LIN {X -0.071,Y -362.649,Z 1312.127,A 0.000,B 0.000,C 90.000,E1 238.869} C_DIS
LIN {X -0.108,Y -362.653,Z 1312.127,A 0.000,B 0.000,C 90.000,E1 238.869} C_DIS
LIN {X -0.177,Y -374.472,Z 1312.111,A 0.000,B 0.000,C 90.000,E1 236.087} C_DIS
LIN {X 0.011,Y -387.676,Z 1312.096,A 0.000,B 0.000,C 90.000,E1 233.336} C_DIS
LIN {X 0.004,Y -402.405,Z 1312.082,A 0.000,B 0.000,C 90.000,E1 230.678} C_DIS
LIN {X 0.038,Y -418.775,Z 1312.067,A 0.000,B 0.000,C 90.000,E1 228.081} C_DIS
LIN {X -0.027,Y -436.906,Z 1312.053,A 0.000,B 0.000,C 90.000,E1 225.567} C_DIS
LIN {X -0.154,Y -444.673,Z 1312.048,A 0.000,B 0.000,C 90.000,E1 224.595} C_DIS
LIN {X -0.168,Y -445.603,Z 1312.047,A 0.000,B 0.000,C 90.000,E1 224.433} C_DIS
LIN {X -0.184,Y -446.772,Z 1312.045,A 0.000,B 0.000,C 90.000,E1 224.109} C_DIS
LIN {X -0.199,Y -447.568,Z 1312.043,A 0.000,B 0.000,C 90.000,E1 223.785} C_DIS
LIN {X 0.112,Y -448.651,Z 1312.040,A 0.000,B 0.000,C 90.000,E1 223.095} C_DIS
LIN {X 0.104,Y -449.370,Z 1312.036,A 0.000,B 0.000,C 90.000,E1 222.447} C_DIS
LIN {X -0.202,Y -449.855,Z 1312.032,A 0.000,B 0.000,C 90.000,E1 221.838} C_DIS
LIN {X -0.168,Y -450.246,Z 1312.025,A 0.000,B 0.000,C 90.000,E1 220.539} C_DIS
LIN {X 0.169,Y -452.965,Z 1312.002,A 0.000,B 0.000,C 90.000,E1 216.297} C_DIS
LIN {X -0.050,Y -454.940,Z 1311.989,A 0.000,B 0.000,C 90.000,E1 214.072} C_DIS
LIN {X 0.055,Y -456.951,Z 1311.979,A 0.000,B 0.000,C 90.000,E1 212.133} C_DIS
LIN {X -0.162,Y -460.306,Z 1311.963,A 0.000,B 0.000,C 90.000,E1 209.283} C_DIS
LIN {X 0.239,Y -462.368,Z 1311.954,A 0.000,B 0.000,C 90.000,E1 207.641} C_DIS
LIN {X -0.160,Y -464.683,Z 1311.945,A 0.000,B 0.000,C 90.000,E1 206.104} C_DIS
LIN {X -0.162,Y -467.452,Z 1311.934,A 0.000,B 0.000,C 90.000,E1 204.207} C_DIS
LIN {X -0.141,Y -468.790,Z 1311.929,A 0.000,B 0.000,C 90.000,E1 203.259} C_DIS
LIN {X 0.099,Y -470.556,Z 1311.922,A 0.000,B 0.000,C 90.000,E1 201.972} C_DIS
LIN {X -0.177,Y -473.597,Z 1311.910,A 0.000,B 0.000,C 90.000,E1 199.812} C_DIS
LIN {X 0.200,Y -476.765,Z 1311.898,A 0.000,B 0.000,C 90.000,E1 197.583} C_DIS
LIN {X 0.067,Y -479.940,Z 1311.886,A 0.000,B 0.000,C 90.000,E1 195.426} C_DIS
LIN {X -0.105,Y -482.521,Z 1311.875,A 0.000,B 0.000,C 90.000,E1 193.592} C_DIS
LIN {X 0.143,Y -485.125,Z 1311.865,A 0.000,B 0.000,C 90.000,E1 191.715} C_DIS
LIN {X -0.123,Y -487.671,Z 1311.855,A 0.000,B 0.000,C 90.000,E1 189.905} C_DIS
LIN {X 0.179,Y -489.766,Z 1311.847,A 0.000,B 0.000,C 90.000,E1 188.341} C_DIS
LIN {X 0.034,Y -491.795,Z 1311.838,A 0.000,B 0.000,C 90.000,E1 186.834} C_DIS
LIN {X -0.032,Y -493.392,Z 1311.831,A 0.000,B 0.000,C 90.000,E1 185.625} C_DIS
LIN {X -0.072,Y -494.846,Z 1311.825,A 0.000,B 0.000,C 90.000,E1 184.416} C_DIS
LIN {X -0.240,Y -496.525,Z 1311.816,A 0.000,B 0.000,C 90.000,E1 182.922} C_DIS
LIN {X -0.045,Y -498.194,Z 1311.806,A 0.000,B 0.000,C 90.000,E1 181.088} C_DIS
LIN {X -0.065,Y -499.139,Z 1311.799,A 0.000,B 0.000,C 90.000,E1 179.885} C_DIS
LIN {X -0.197,Y -499.875,Z 1311.791,A 0.000,B 0.000,C 90.000,E1 178.396} C_DIS
LIN {X 0.068,Y -500.147,Z 1311.788,A 0.000,B 0.000,C 90.000,E1 177.764} C_DIS
LIN {X -0.035,Y -500.371,Z 1311.779,A 0.000,B 0.000,C 90.000,E1 176.274} C_DIS
LIN {X 0.114,Y -500.298,Z 1311.774,A 0.000,B 0.000,C 90.000,E1 175.355} C_DIS
LIN {X -0.107,Y -500.165,Z 1311.771,A 0.000,B 0.000,C 90.000,E1 174.780} C_DIS
LIN {X -0.053,Y -499.594,Z 1311.764,A 0.000,B 0.000,C 90.000,E1 173.571} C_DIS
LIN {X 0.133,Y -499.048,Z 1311.759,A 0.000,B 0.000,C 90.000,E1 172.648} C_DIS
LIN {X -0.182,Y -498.189,Z 1311.754,A 0.000,B 0.000,C 90.000,E1 171.781} C_DIS
LIN {X 0.062,Y -496.946,Z 1311.749,A 0.000,B 0.000,C 90.000,E1 170.849} C_DIS
LIN {X 0.211,Y -495.510,Z 1311.744,A 0.000,B 0.000,C 90.000,E1 169.926} C_DIS
LIN {X -0.061,Y -493.810,Z 1311.739,A 0.000,B 0.000,C 90.000,E1 169.050} C_DIS
LIN {X 0.031,Y -490.996,Z 1311.732,A 0.000,B 0.000,C 90.000,E1 167.825} C_DIS
LIN {X -0.073,Y -489.328,Z 1311.729,A 0.000,B 0.000,C 90.000,E1 167.229} C_DIS
LIN {X 0.062,Y -486.673,Z 1311.724,A 0.000,B 0.000,C 90.000,E1 166.297} C_DIS
LIN {X 0.264,Y -482.251,Z 1311.717,A 0.000,B 0.000,C 90.000,E1 165.046} C_DIS
LIN {X 0.175,Y -477.177,Z 1311.711,A 0.000,B 0.000,C 90.000,E1 163.976} C_DIS
LIN {X -0.190,Y -472.157,Z 1311.706,A 0.000,B 0.000,C 90.000,E1 163.087} C_DIS
LIN {X -0.145,Y -463.602,Z 1311.697,A 0.000,B 0.000,C 90.000,E1 161.511} C_DIS
LIN {X -0.178,Y -461.464,Z 1311.695,A 0.000,B 0.000,C 90.000,E1 161.040} C_DIS
LIN {X 0.099,Y -459.056,Z 1311.691,A 0.000,B 0.000,C 90.000,E1 160.369} C_DIS
LIN {X -0.070,Y -457.395,Z 1311.688,A 0.000,B 0.000,C 90.000,E1 159.752} C_DIS
LIN {X -0.080,Y -456.796,Z 1311.683,A 0.000,B 0.000,C 90.000,E1 158.954} C_DIS
LIN {X 0.087,Y -456.802,Z 1311.682,A 0.000,B 0.000,C 90.000,E1 158.773} C_DIS
LIN {X 0.170,Y -457.421,Z 1311.680,A 0.000,B 0.000,C 90.000,E1 158.411} C_DIS
LIN {X 0.130,Y -457.459,Z 1311.680,A 0.000,B 0.000,C 90.000,E1 158.411} C_DIS
LIN {X -0.163,Y -459.940,Z 1311.678,A 0.000,B 0.000,C 90.000,E1 158.103} C_DIS
LIN {X 0.005,Y -463.307,Z 1311.677,A 0.000,B 0.000,C 90.000,E1 157.794} C_DIS
LIN {X -0.102,Y -466.278,Z 1311.675,A 0.000,B 0.000,C 90.000,E1 157.539} C_DIS
LIN {X 0.005,Y -482.916,Z 1311.668,A 0.000,B 0.000,C 90.000,E1 156.177} C_DIS
LIN {X 0.207,Y -490.314,Z 1311.664,A 0.000,B 0.000,C 90.000,E1 155.537} C_DIS
LIN {X 0.022,Y -494.675,Z 1311.662,A 0.000,B 0.000,C 90.000,E1 155.177} C_DIS
LIN {X -0.251,Y -502.876,Z 1311.658,A 0.000,B 0.000,C 90.000,E1 154.409} C_DIS
LIN {X -0.051,Y -506.911,Z 1311.655,A 0.000,B 0.000,C 90.000,E1 153.973} C_DIS
LIN {X 0.132,Y -512.097,Z 1311.652,A 0.000,B 0.000,C 90.000,E1 153.384} C_DIS
LIN {X 0.128,Y -515.865,Z 1311.650,A 0.000,B 0.000,C 90.000,E1 152.948} C_DIS
LIN {X -0.149,Y -519.429,Z 1311.647,A 0.000,B 0.000,C 90.000,E1 152.538} C_DIS
LIN {X -0.104,Y -523.631,Z 1311.644,A 0.000,B 0.000,C 90.000,E1 151.948} C_DIS
LIN {X -0.278,Y -527.388,Z 1311.641,A 0.000,B 0.000,C 90.000,E1 151.385} C_DIS
LIN {X -0.070,Y -531.210,Z 1311.637,A 0.000,B 0.000,C 90.000,E1 150.639} C_DIS
LIN {X -0.201,Y -533.675,Z 1311.634,A 0.000,B 0.000,C 90.000,E1 150.078} C_DIS
LIN {X 0.217,Y -535.635,Z 1311.630,A 0.000,B 0.000,C 90.000,E1 149.459} C_DIS
LIN {X -0.073,Y -536.553,Z 1311.629,A 0.000,B 0.000,C 90.000,E1 149.203} C_DIS
LIN {X 0.093,Y -538.129,Z 1311.626,A 0.000,B 0.000,C 90.000,E1 148.614} C_DIS
LIN {X -0.187,Y -540.015,Z 1311.621,A 0.000,B 0.000,C 90.000,E1 147.788} C_DIS
LIN {X -0.001,Y -541.094,Z 1311.618,A 0.000,B 0.000,C 90.000,E1 147.199} C_DIS
LIN {X 0.052,Y -542.385,Z 1311.613,A 0.000,B 0.000,C 90.000,E1 146.342} C_DIS
LIN {X 0.333,Y -544.220,Z 1311.605,A 0.000,B 0.000,C 90.000,E1 144.895} C_DIS
LIN {X 0.084,Y -544.934,Z 1311.602,A 0.000,B 0.000,C 90.000,E1 144.356} C_DIS
LIN {X -0.181,Y -546.138,Z 1311.599,A 0.000,B 0.000,C 90.000,E1 143.783} C_DIS
LIN {X -0.223,Y -546.147,Z 1311.599,A 0.000,B 0.000,C 90.000,E1 143.783} C_DIS
LIN {X 0.337,Y -546.727,Z 1311.598,A 0.000,B 0.000,C 90.000,E1 143.623} C_DIS
LIN {X 0.195,Y -548.575,Z 1311.597,A 0.000,B 0.000,C 90.000,E1 143.497} C_DIS
LIN {X -0.128,Y -550.841,Z 1311.597,A 0.000,B 0.000,C 90.000,E1 143.417} C_DIS
LIN {X 0.072,Y -560.861,Z 1311.595,A 0.000,B 0.000,C 90.000,E1 143.050} C_DIS
LIN {X 0.300,Y -566.988,Z 1311.593,A 0.000,B 0.000,C 90.000,E1 142.763} C_DIS
LIN {X 0.093,Y -573.111,Z 1311.592,A 0.000,B 0.000,C 90.000,E1 142.477} C_DIS
LIN {X 0.094,Y -580.448,Z 1311.589,A 0.000,B 0.000,C 90.000,E1 142.029} C_DIS
LIN {X 0.232,Y -586.267,Z 1311.587,A 0.000,B 0.000,C 90.000,E1 141.618} C_DIS
LIN {X 0.106,Y -590.462,Z 1311.585,A 0.000,B 0.000,C 90.000,E1 141.295} C_DIS
LIN {X 0.001,Y -594.417,Z 1311.583,A 0.000,B 0.000,C 90.000,E1 140.964} C_DIS
LIN {X -0.084,Y -599.469,Z 1311.580,A 0.000,B 0.000,C 90.000,E1 140.481} C_DIS
LIN {X 0.187,Y -603.081,Z 1311.578,A 0.000,B 0.000,C 90.000,E1 140.070} C_DIS
LIN {X 0.243,Y -607.562,Z 1311.575,A 0.000,B 0.000,C 90.000,E1 139.542} C_DIS
LIN {X -0.207,Y -612.712,Z 1311.572,A 0.000,B 0.000,C 90.000,E1 138.933} C_DIS
LIN {X -0.101,Y -616.473,Z 1311.569,A 0.000,B 0.000,C 90.000,E1 138.405} C_DIS
LIN {X -0.070,Y -620.894,Z 1311.565,A 0.000,B 0.000,C 90.000,E1 137.757} C_DIS
LIN {X 0.083,Y -625.633,Z 1311.561,A 0.000,B 0.000,C 90.000,E1 136.986} C_DIS
LIN {X -0.230,Y -629.505,Z 1311.558,A 0.000,B 0.000,C 90.000,E1 136.377} C_DIS
LIN {X 0.106,Y -636.631,Z 1311.551,A 0.000,B 0.000,C 90.000,E1 135.081} C_DIS
LIN {X -0.085,Y -639.363,Z 1311.548,A 0.000,B 0.000,C 90.000,E1 134.595} C_DIS
LIN {X 0.075,Y -644.084,Z 1311.543,A 0.000,B 0.000,C 90.000,E1 133.704} C_DIS
LIN {X -0.277,Y -651.221,Z 1311.535,A 0.000,B 0.000,C 90.000,E1 132.366} C_DIS
LIN {X 0.029,Y -656.976,Z 1311.529,A 0.000,B 0.000,C 90.000,E1 131.229} C_DIS
LIN {X -0.036,Y -661.842,Z 1311.524,A 0.000,B 0.000,C 90.000,E1 130.253} C_DIS
LIN {X -0.045,Y -666.291,Z 1311.518,A 0.000,B 0.000,C 90.000,E1 129.277} C_DIS
LIN {X -0.004,Y -670.441,Z 1311.513,A 0.000,B 0.000,C 90.000,E1 128.302} C_DIS
LIN {X 0.085,Y -673.306,Z 1311.509,A 0.000,B 0.000,C 90.000,E1 127.569} C_DIS
LIN {X 0.333,Y -676.851,Z 1311.503,A 0.000,B 0.000,C 90.000,E1 126.583} C_DIS
LIN {X 0.083,Y -679.216,Z 1311.499,A 0.000,B 0.000,C 90.000,E1 125.884} C_DIS
LIN {X -0.140,Y -682.074,Z 1311.494,A 0.000,B 0.000,C 90.000,E1 124.945} C_DIS
LIN {X 0.219,Y -684.041,Z 1311.490,A 0.000,B 0.000,C 90.000,E1 124.199} C_DIS
LIN {X -0.341,Y -686.371,Z 1311.485,A 0.000,B 0.000,C 90.000,E1 123.293} C_DIS
LIN {X -0.303,Y -688.375,Z 1311.480,A 0.000,B 0.000,C 90.000,E1 122.339} C_DIS
LIN {X -0.017,Y -690.462,Z 1311.473,A 0.000,B 0.000,C 90.000,E1 121.131} C_DIS
LIN {X -0.283,Y -691.849,Z 1311.468,A 0.000,B 0.000,C 90.000,E1 120.207} C_DIS
LIN {X 0.172,Y -692.835,Z 1311.464,A 0.000,B 0.000,C 90.000,E1 119.461} C_DIS
LIN {X -0.070,Y -693.840,Z 1311.459,A 0.000,B 0.000,C 90.000,E1 118.537} C_DIS
LIN {X -0.016,Y -694.350,Z 1311.453,A 0.000,B 0.000,C 90.000,E1 117.590} C_DIS
LIN {X 0.374,Y -694.631,Z 1311.448,A 0.000,B 0.000,C 90.000,E1 116.616} C_DIS
LIN {X 0.202,Y -694.499,Z 1311.444,A 0.000,B 0.000,C 90.000,E1 115.924} C_DIS
LIN {X 0.079,Y -694.301,Z 1311.442,A 0.000,B 0.000,C 90.000,E1 115.463} C_DIS
LIN {X -0.343,Y -693.843,Z 1311.439,A 0.000,B 0.000,C 90.000,E1 115.027} C_DIS
LIN {X 0.153,Y -693.130,Z 1311.436,A 0.000,B 0.000,C 90.000,E1 114.515} C_DIS
LIN {X 0.113,Y -692.603,Z 1311.435,A 0.000,B 0.000,C 90.000,E1 114.283} C_DIS
LIN {X -0.032,Y -691.135,Z 1311.432,A 0.000,B 0.000,C 90.000,E1 113.823} C_DIS
LIN {X 0.163,Y -688.532,Z 1311.430,A 0.000,B 0.000,C 90.000,E1 113.334} C_DIS
LIN {X 0.277,Y -687.855,Z 1311.429,A 0.000,B 0.000,C 90.000,E1 113.206} C_DIS
LIN {X -0.242,Y -686.910,Z 1311.428,A 0.000,B 0.000,C 90.000,E1 113.131} C_DIS
LIN {X 0.266,Y -681.553,Z 1311.426,A 0.000,B 0.000,C 90.000,E1 112.642} C_DIS
LIN {X -0.175,Y -679.920,Z 1311.425,A 0.000,B 0.000,C 90.000,E1 112.567} C_DIS
LIN {X -0.184,Y -675.396,Z 1311.424,A 0.000,B 0.000,C 90.000,E1 112.386} C_DIS
LIN {X 0.245,Y -673.452,Z 1311.424,A 0.000,B 0.000,C 90.000,E1 112.280} C_DIS
LIN {X -0.220,Y -666.520,Z 1311.423,A 0.000,B 0.000,C 90.000,E1 112.153} C_DIS
LIN {X 0.113,Y -663.945,Z 1311.423,A 0.000,B 0.000,C 90.000,E1 112.078} C_DIS
LIN {X -0.282,Y -655.505,Z 1311.422,A 0.000,B 0.000,C 90.000,E1 112.025} C_DIS
LIN {X 0.065,Y -649.452,Z 1311.422,A 0.000,B 0.000,C 90.000,E1 111.972} C_DIS
LIN {X 0.258,Y -645.085,Z 1311.422,A 0.000,B 0.000,C 90.000,E1 111.897} C_DIS
LIN {X -0.024,Y -643.791,Z 1311.422,A 0.000,B 0.000,C 90.000,E1 111.897} C_DIS
LIN {X -0.078,Y -642.090,Z 1311.421,A 0.000,B 0.000,C 90.000,E1 111.844} C_DIS
LIN {X -0.119,Y -642.053,Z 1311.421,A 0.000,B 0.000,C 90.000,E1 111.844} C_DIS
LIN {X -0.156,Y -643.053,Z 1311.420,A 0.000,B 0.000,C 90.000,E1 111.642} C_DIS
LIN {X 0.244,Y -645.869,Z 1311.418,A 0.000,B 0.000,C 90.000,E1 111.227} C_DIS
LIN {X 0.229,Y -651.693,Z 1311.414,A 0.000,B 0.000,C 90.000,E1 110.482} C_DIS
LIN {X -0.008,Y -655.900,Z 1311.411,A 0.000,B 0.000,C 90.000,E1 109.885} C_DIS
LIN {X 0.015,Y -659.535,Z 1311.407,A 0.000,B 0.000,C 90.000,E1 109.268} C_DIS
LIN {X -0.153,Y -662.652,Z 1311.404,A 0.000,B 0.000,C 90.000,E1 108.671} C_DIS
LIN {X -0.237,Y -665.922,Z 1311.400,A 0.000,B 0.000,C 90.000,E1 107.946} C_DIS
LIN {X -0.294,Y -668.770,Z 1311.396,A 0.000,B 0.000,C 90.000,E1 107.221} C_DIS
LIN {X -0.254,Y -670.453,Z 1311.393,A 0.000,B 0.000,C 90.000,E1 106.732} C_DIS
LIN {X 0.183,Y -672.621,Z 1311.389,A 0.000,B 0.000,C 90.000,E1 105.969} C_DIS
LIN {X 0.183,Y -674.414,Z 1311.385,A 0.000,B 0.000,C 90.000,E1 105.245} C_DIS
LIN {X 0.018,Y -675.919,Z 1311.381,A 0.000,B 0.000,C 90.000,E1 104.537} C_DIS
LIN {X -0.131,Y -677.197,Z 1311.377,A 0.000,B 0.000,C 90.000,E1 103.828} C_DIS
LIN {X -0.269,Y -677.981,Z 1311.373,A 0.000,B 0.000,C 90.000,E1 103.119} C_DIS
LIN {X 0.260,Y -678.463,Z 1311.369,A 0.000,B 0.000,C 90.000,E1 102.355} C_DIS
LIN {X 0.171,Y -678.639,Z 1311.366,A 0.000,B 0.000,C 90.000,E1 101.883} C_DIS
LIN {X -0.053,Y -678.589,Z 1311.364,A 0.000,B 0.000,C 90.000,E1 101.422} C_DIS
LIN {X -0.188,Y -678.054,Z 1311.359,A 0.000,B 0.000,C 90.000,E1 100.715} C_DIS
LIN {X 0.259,Y -677.529,Z 1311.357,A 0.000,B 0.000,C 90.000,E1 100.197} C_DIS
LIN {X 0.156,Y -676.732,Z 1311.354,A 0.000,B 0.000,C 90.000,E1 99.726} C_DIS
LIN {X -0.068,Y -675.668,Z 1311.351,A 0.000,B 0.000,C 90.000,E1 99.265} C_DIS
LIN {X -0.292,Y -674.222,Z 1311.349,A 0.000,B 0.000,C 90.000,E1 98.803} C_DIS
LIN {X 0.072,Y -671.486,Z 1311.345,A 0.000,B 0.000,C 90.000,E1 98.049} C_DIS
LIN {X -0.258,Y -668.089,Z 1311.341,A 0.000,B 0.000,C 90.000,E1 97.352} C_DIS
LIN {X 0.135,Y -665.537,Z 1311.338,A 0.000,B 0.000,C 90.000,E1 96.834} C_DIS
LIN {X -0.336,Y -661.432,Z 1311.334,A 0.000,B 0.000,C 90.000,E1 96.144} C_DIS
LIN {X -0.087,Y -657.553,Z 1311.331,A 0.000,B 0.000,C 90.000,E1 95.511} C_DIS
LIN {X 0.128,Y -653.294,Z 1311.327,A 0.000,B 0.000,C 90.000,E1 94.878} C_DIS
LIN {X -0.235,Y -649.570,Z 1311.324,A 0.000,B 0.000,C 90.000,E1 94.416} C_DIS
LIN {X -0.091,Y -644.408,Z 1311.321,A 0.000,B 0.000,C 90.000,E1 93.784} C_DIS
LIN {X -0.030,Y -638.855,Z 1311.318,A 0.000,B 0.000,C 90.000,E1 93.154} C_DIS
LIN {X -0.094,Y -631.872,Z 1311.313,A 0.000,B 0.000,C 90.000,E1 92.407} C_DIS
LIN {X 0.015,Y -625.689,Z 1311.310,A 0.000,B 0.000,C 90.000,E1 91.776} C_DIS
LIN {X -0.275,Y -620.348,Z 1311.307,A 0.000,B 0.000,C 90.000,E1 91.318} C_DIS
LIN {X 0.254,Y -616.296,Z 1311.305,A 0.000,B 0.000,C 90.000,E1 90.917} C_DIS
LIN {X 0.010,Y -608.830,Z 1311.302,A 0.000,B 0.000,C 90.000,E1 90.401} C_DIS
LIN {X 0.226,Y -602.513,Z 1311.300,A 0.000,B 0.000,C 90.000,E1 90.000} C_DIS
LIN {X 0.163,Y -595.886,Z 1311.298,A 0.000,B 0.000,C 90.000,E1 89.656} C_DIS
LIN {X -0.081,Y -588.867,Z 1311.297,A 0.000,B 0.000,C 90.000,E1 89.370} C_DIS
LIN {X -0.101,Y -576.659,Z 1311.294,A 0.000,B 0.000,C 90.000,E1 88.912} C_DIS
LIN {X -0.178,Y -572.876,Z 1311.293,A 0.000,B 0.000,C 90.000,E1 88.740} C_DIS
LIN {X -0.217,Y -572.799,Z 1311.293,A 0.000,B 0.000,C 90.000,E1 88.740} C_DIS
LIN {X 0.199,Y -570.811,Z 1311.292,A 0.000,B 0.000,C 90.000,E1 88.453} C_DIS
LIN {X 0.156,Y -570.803,Z 1311.292,A 0.000,B 0.000,C 90.000,E1 88.453} C_DIS
LIN {X 0.144,Y -570.501,Z 1311.290,A 0.000,B 0.000,C 90.000,E1 88.224} C_DIS
LIN {X 0.053,Y -570.697,Z 1311.287,A 0.000,B 0.000,C 90.000,E1 87.650} C_DIS
LIN {X 0.035,Y -571.783,Z 1311.281,A 0.000,B 0.000,C 90.000,E1 86.560} C_DIS
LIN {X -0.173,Y -574.648,Z 1311.266,A 0.000,B 0.000,C 90.000,E1 83.856} C_DIS
LIN {X 0.204,Y -577.511,Z 1311.252,A 0.000,B 0.000,C 90.000,E1 81.376} C_DIS
LIN {X 0.264,Y -579.450,Z 1311.243,A 0.000,B 0.000,C 90.000,E1 79.746} C_DIS
LIN {X 0.136,Y -580.891,Z 1311.236,A 0.000,B 0.000,C 90.000,E1 78.409} C_DIS
LIN {X -0.194,Y -582.408,Z 1311.227,A 0.000,B 0.000,C 90.000,E1 76.825} C_DIS
LIN {X -0.025,Y -583.440,Z 1311.219,A 0.000,B 0.000,C 90.000,E1 75.463} C_DIS
LIN {X -0.068,Y -584.221,Z 1311.213,A 0.000,B 0.000,C 90.000,E1 74.393} C_DIS
LIN {X 0.127,Y -585.071,Z 1311.206,A 0.000,B 0.000,C 90.000,E1 73.032} C_DIS
LIN {X -0.207,Y -586.113,Z 1311.197,A 0.000,B 0.000,C 90.000,E1 71.456} C_DIS
LIN {X 0.040,Y -587.148,Z 1311.188,A 0.000,B 0.000,C 90.000,E1 69.826} C_DIS
LIN {X -0.048,Y -588.218,Z 1311.179,A 0.000,B 0.000,C 90.000,E1 68.230} C_DIS
LIN {X -0.319,Y -589.132,Z 1311.172,A 0.000,B 0.000,C 90.000,E1 66.922} C_DIS
LIN {X -0.006,Y -590.407,Z 1311.161,A 0.000,B 0.000,C 90.000,E1 65.025} C_DIS
LIN {X -0.187,Y -591.697,Z 1311.151,A 0.000,B 0.000,C 90.000,E1 63.179} C_DIS
LIN {X -0.172,Y -593.530,Z 1311.139,A 0.000,B 0.000,C 90.000,E1 61.051} C_DIS
LIN {X -0.046,Y -595.600,Z 1311.127,A 0.000,B 0.000,C 90.000,E1 58.918} C_DIS
LIN {X 0.227,Y -597.569,Z 1311.117,A 0.000,B 0.000,C 90.000,E1 57.041} C_DIS
LIN {X -0.110,Y -598.989,Z 1311.110,A 0.000,B 0.000,C 90.000,E1 55.754} C_DIS
LIN {X 0.009,Y -600.062,Z 1311.104,A 0.000,B 0.000,C 90.000,E1 54.689} C_DIS
LIN {X -0.195,Y -601.500,Z 1311.095,A 0.000,B 0.000,C 90.000,E1 53.130} C_DIS
LIN {X -0.009,Y -602.810,Z 1311.086,A 0.000,B 0.000,C 90.000,E1 51.537} C_DIS
LIN {X -0.019,Y -604.099,Z 1311.076,A 0.000,B 0.000,C 90.000,E1 49.703} C_DIS
LIN {X -0.178,Y -604.564,Z 1311.072,A 0.000,B 0.000,C 90.000,E1 48.933} C_DIS
LIN {X -0.079,Y -604.890,Z 1311.066,A 0.000,B 0.000,C 90.000,E1 47.877} C_DIS
LIN {X -0.160,Y -605.118,Z 1311.056,A 0.000,B 0.000,C 90.000,E1 46.053} C_DIS
LIN {X -0.082,Y -605.165,Z 1311.050,A 0.000,B 0.000,C 90.000,E1 45.000} C_DIS
LIN {X -0.003,Y -605.019,Z 1311.044,A 0.000,B 0.000,C 90.000,E1 43.947} C_DIS
LIN {X 0.113,Y -604.567,Z 1311.036,A 0.000,B 0.000,C 90.000,E1 42.366} C_DIS
LIN {X 0.011,Y -604.123,Z 1311.028,A 0.000,B 0.000,C 90.000,E1 41.067} C_DIS
LIN {X 0.107,Y -603.633,Z 1311.022,A 0.000,B 0.000,C 90.000,E1 40.011} C_DIS
LIN {X -0.188,Y -603.162,Z 1311.017,A 0.000,B 0.000,C 90.000,E1 38.991} C_DIS
LIN {X 0.107,Y -602.673,Z 1311.012,A 0.000,B 0.000,C 90.000,E1 38.177} C_DIS
LIN {X 0.026,Y -602.049,Z 1311.008,A 0.000,B 0.000,C 90.000,E1 37.397} C_DIS
LIN {X -0.288,Y -600.957,Z 1311.002,A 0.000,B 0.000,C 90.000,E1 36.377} C_DIS
LIN {X 0.104,Y -599.106,Z 1310.995,A 0.000,B 0.000,C 90.000,E1 35.025} C_DIS
LIN {X -0.119,Y -597.290,Z 1310.989,A 0.000,B 0.000,C 90.000,E1 33.992} C_DIS
LIN {X 0.238,Y -595.709,Z 1310.984,A 0.000,B 0.000,C 90.000,E1 33.166} C_DIS
LIN {X -0.246,Y -593.925,Z 1310.980,A 0.000,B 0.000,C 90.000,E1 32.418} C_DIS
LIN {X 0.070,Y -591.876,Z 1310.976,A 0.000,B 0.000,C 90.000,E1 31.592} C_DIS
LIN {X 0.051,Y -589.439,Z 1310.971,A 0.000,B 0.000,C 90.000,E1 30.797} C_DIS
LIN {X 0.125,Y -587.679,Z 1310.968,A 0.000,B 0.000,C 90.000,E1 30.256} C_DIS
LIN {X 0.062,Y -584.645,Z 1310.964,A 0.000,B 0.000,C 90.000,E1 29.461} C_DIS
LIN {X -0.186,Y -582.373,Z 1310.961,A 0.000,B 0.000,C 90.000,E1 28.949} C_DIS
LIN {X 0.205,Y -578.708,Z 1310.956,A 0.000,B 0.000,C 90.000,E1 28.103} C_DIS
LIN {X 0.038,Y -574.503,Z 1310.952,A 0.000,B 0.000,C 90.000,E1 27.308} C_DIS
LIN {X 0.153,Y -570.702,Z 1310.948,A 0.000,B 0.000,C 90.000,E1 26.616} C_DIS
LIN {X 0.153,Y -565.727,Z 1310.943,A 0.000,B 0.000,C 90.000,E1 25.796} C_DIS
LIN {X -0.308,Y -561.156,Z 1310.940,A 0.000,B 0.000,C 90.000,E1 25.155} C_DIS
LIN {X -0.096,Y -558.238,Z 1310.937,A 0.000,B 0.000,C 90.000,E1 24.719} C_DIS
LIN {X -0.112,Y -552.956,Z 1310.933,A 0.000,B 0.000,C 90.000,E1 24.027} C_DIS
LIN {X -0.166,Y -547.401,Z 1310.930,A 0.000,B 0.000,C 90.000,E1 23.334} C_DIS
LIN {X 0.098,Y -540.177,Z 1310.925,A 0.000,B 0.000,C 90.000,E1 22.461} C_DIS
LIN {X -0.085,Y -533.890,Z 1310.921,A 0.000,B 0.000,C 90.000,E1 21.770} C_DIS
LIN {X 0.239,Y -522.221,Z 1310.914,A 0.000,B 0.000,C 90.000,E1 20.482} C_DIS
LIN {X 0.115,Y -512.971,Z 1310.909,A 0.000,B 0.000,C 90.000,E1 19.523} C_DIS
LIN {X 0.023,Y -501.882,Z 1310.902,A 0.000,B 0.000,C 90.000,E1 18.417} C_DIS
LIN {X 0.151,Y -490.858,Z 1310.896,A 0.000,B 0.000,C 90.000,E1 17.330} C_DIS
LIN {X -0.160,Y -483.700,Z 1310.893,A 0.000,B 0.000,C 90.000,E1 16.677} C_DIS
LIN {X 0.078,Y -476.334,Z 1310.889,A 0.000,B 0.000,C 90.000,E1 15.969} C_DIS
LIN {X 0.109,Y -464.557,Z 1310.883,A 0.000,B 0.000,C 90.000,E1 14.898} C_DIS
LIN {X -0.185,Y -442.753,Z 1310.871,A 0.000,B 0.000,C 90.000,E1 12.883} C_DIS
LIN {X -0.129,Y -424.029,Z 1310.861,A 0.000,B 0.000,C 90.000,E1 10.950} C_DIS
LIN {X 0.003,Y -409.779,Z 1310.852,A 0.000,B 0.000,C 90.000,E1 9.378} C_DIS
LIN {X 0.171,Y -401.165,Z 1310.847,A 0.000,B 0.000,C 90.000,E1 8.398} C_DIS
LIN {X -0.089,Y -398.370,Z 1310.845,A 0.000,B 0.000,C 90.000,E1 8.106} C_DIS
LIN {X -0.074,Y -395.420,Z 1310.842,A 0.000,B 0.000,C 90.000,E1 7.644} C_DIS
LIN {X -0.112,Y -395.442,Z 1310.842,A 0.000,B 0.000,C 90.000,E1 7.644} C_DIS
LIN {X 0.154,Y -396.271,Z 1310.842,A 0.000,B 0.000,C 90.000,E1 7.473} C_DIS
LIN {X 0.018,Y -400.435,Z 1310.840,A 0.000,B 0.000,C 90.000,E1 7.125} C_DIS
LIN {X 0.136,Y -408.992,Z 1310.837,A 0.000,B 0.000,C 90.000,E1 6.549} C_DIS
LIN {X 0.088,Y -417.236,Z 1310.834,A 0.000,B 0.000,C 90.000,E1 6.030} C_DIS
LIN {X 0.145,Y -423.721,Z 1310.831,A 0.000,B 0.000,C 90.000,E1 5.568} C_DIS
LIN {X -0.158,Y -433.047,Z 1310.827,A 0.000,B 0.000,C 90.000,E1 4.878} C_DIS
LIN {X 0.123,Y -442.041,Z 1310.823,A 0.000,B 0.000,C 90.000,E1 4.073} C_DIS
LIN {X -0.030,Y -450.911,Z 1310.818,A 0.000,B 0.000,C 90.000,E1 3.269} C_DIS
LIN {X 0.227,Y -458.153,Z 1310.814,A 0.000,B 0.000,C 90.000,E1 2.522} C_DIS
LIN {X -0.029,Y -462.248,Z 1310.812,A 0.000,B 0.000,C 90.000,E1 2.121} C_DIS
LIN {X 0.088,Y -466.383,Z 1310.809,A 0.000,B 0.000,C 90.000,E1 1.661} C_DIS
LIN {X 0.194,Y -472.544,Z 1310.805,A 0.000,B 0.000,C 90.000,E1 0.917} C_DIS
LIN {X -0.084,Y -478.505,Z 1310.801,A 0.000,B 0.000,C 90.000,E1 0.172} C_DIS
LIN {X 0.138,Y -484.372,Z 1310.796,A 0.000,B 0.000,C 90.000,E1 359.312} C_DIS
LIN {X -0.062,Y -489.328,Z 1310.792,A 0.000,B 0.000,C 90.000,E1 358.568} C_DIS
LIN {X -0.202,Y -493.919,Z 1310.788,A 0.000,B 0.000,C 90.000,E1 357.822} C_DIS
LIN {X -0.001,Y -497.459,Z 1310.784,A 0.000,B 0.000,C 90.000,E1 357.192} C_DIS
LIN {X 0.124,Y -502.221,Z 1310.779,A 0.000,B 0.000,C 90.000,E1 356.274} C_DIS
LIN {X 0.109,Y -505.946,Z 1310.775,A 0.000,B 0.000,C 90.000,E1 355.527} C_DIS
LIN {X 0.130,Y -509.406,Z 1310.771,A 0.000,B 0.000,C 90.000,E1 354.780} C_DIS
LIN {X 0.139,Y -513.978,Z 1310.765,A 0.000,B 0.000,C 90.000,E1 353.742} C_DIS
LIN {X 0.013,Y -516.372,Z 1310.762,A 0.000,B 0.000,C 90.000,E1 353.166} C_DIS
LIN {X -0.115,Y -519.623,Z 1310.757,A 0.000,B 0.000,C 90.000,E1 352.299} C_DIS
LIN {X -0.210,Y -522.596,Z 1310.752,A 0.000,B 0.000,C 90.000,E1 351.432} C_DIS
LIN {X -0.202,Y -524.397,Z 1310.749,A 0.000,B 0.000,C 90.000,E1 350.849} C_DIS
LIN {X -0.228,Y -527.751,Z 1310.743,A 0.000,B 0.000,C 90.000,E1 349.690} C_DIS
LIN {X -0.148,Y -530.014,Z 1310.738,A 0.000,B 0.000,C 90.000,E1 348.814} C_DIS
LIN {X -0.079,Y -531.373,Z 1310.735,A 0.000,B 0.000,C 90.000,E1 348.229} C_DIS
LIN {X 0.086,Y -533.805,Z 1310.728,A 0.000,B 0.000,C 90.000,E1 347.061} C_DIS
LIN {X -0.168,Y -535.311,Z 1310.723,A 0.000,B 0.000,C 90.000,E1 346.228} C_DIS
LIN {X 0.178,Y -537.055,Z 1310.717,A 0.000,B 0.000,C 90.000,E1 345.046} C_DIS
LIN {X -0.231,Y -537.771,Z 1310.714,A 0.000,B 0.000,C 90.000,E1 344.519} C_DIS
LIN {X -0.229,Y -538.712,Z 1310.708,A 0.000,B 0.000,C 90.000,E1 343.378} C_DIS
LIN {X 0.092,Y -539.315,Z 1310.703,A 0.000,B 0.000,C 90.000,E1 342.489} C_DIS
LIN {X 0.066,Y -539.488,Z 1310.698,A 0.000,B 0.000,C 90.000,E1 341.638} C_DIS
LIN {X -0.196,Y -539.132,Z 1310.690,A 0.000,B 0.000,C 90.000,E1 340.242} C_DIS
LIN {X 0.065,Y -538.772,Z 1310.687,A 0.000,B 0.000,C 90.000,E1 339.645} C_DIS
LIN {X 0.225,Y -537.970,Z 1310.682,A 0.000,B 0.000,C 90.000,E1 338.773} C_DIS
LIN {X 0.183,Y -536.943,Z 1310.677,A 0.000,B 0.000,C 90.000,E1 337.922} C_DIS
LIN {X 0.117,Y -536.085,Z 1310.674,A 0.000,B 0.000,C 90.000,E1 337.358} C_DIS
LIN {X 0.047,Y -534.907,Z 1310.671,A 0.000,B 0.000,C 90.000,E1 336.794} C_DIS
LIN {X -0.168,Y -534.482,Z 1310.670,A 0.000,B 0.000,C 90.000,E1 336.538} C_DIS
LIN {X -0.045,Y -532.331,Z 1310.665,A 0.000,B 0.000,C 90.000,E1 335.665} C_DIS
LIN {X 0.049,Y -529.897,Z 1310.660,A 0.000,B 0.000,C 90.000,E1 334.793} C_DIS
LIN {X -0.105,Y -524.390,Z 1310.650,A 0.000,B 0.000,C 90.000,E1 333.076} C_DIS
LIN {X 0.044,Y -520.538,Z 1310.644,A 0.000,B 0.000,C 90.000,E1 331.897} C_DIS
LIN {X -0.229,Y -517.521,Z 1310.639,A 0.000,B 0.000,C 90.000,E1 331.051} C_DIS
LIN {X 0.169,Y -514.299,Z 1310.634,A 0.000,B 0.000,C 90.000,E1 330.127} C_DIS
LIN {X 0.002,Y -511.402,Z 1310.630,A 0.000,B 0.000,C 90.000,E1 329.410} C_DIS
LIN {X 0.104,Y -505.146,Z 1310.622,A 0.000,B 0.000,C 90.000,E1 327.916} C_DIS
LIN {X 0.017,Y -499.499,Z 1310.614,A 0.000,B 0.000,C 90.000,E1 326.580} C_DIS
LIN {X -0.235,Y -497.281,Z 1310.611,A 0.000,B 0.000,C 90.000,E1 326.008} C_DIS
LIN {X -0.090,Y -495.617,Z 1310.608,A 0.000,B 0.000,C 90.000,E1 325.388} C_DIS
LIN {X -0.102,Y -493.843,Z 1310.603,A 0.000,B 0.000,C 90.000,E1 324.482} C_DIS
LIN {X 0.010,Y -492.369,Z 1310.596,A 0.000,B 0.000,C 90.000,E1 323.256} C_DIS
LIN {X 0.103,Y -491.341,Z 1310.589,A 0.000,B 0.000,C 90.000,E1 322.029} C_DIS
LIN {X 0.025,Y -490.436,Z 1310.584,A 0.000,B 0.000,C 90.000,E1 321.126} C_DIS
LIN {X 0.018,Y -489.633,Z 1310.581,A 0.000,B 0.000,C 90.000,E1 320.517} C_DIS
LIN {X 0.169,Y -489.102,Z 1310.579,A 0.000,B 0.000,C 90.000,E1 320.194} C_DIS
LIN {X 0.007,Y -488.432,Z 1310.577,A 0.000,B 0.000,C 90.000,E1 319.908} C_DIS
LIN {X -0.158,Y -487.555,Z 1310.576,A 0.000,B 0.000,C 90.000,E1 319.622} C_DIS
LIN {X -0.083,Y -486.987,Z 1310.575,A 0.000,B 0.000,C 90.000,E1 319.461} C_DIS
LIN {X -0.009,Y -486.260,Z 1310.574,A 0.000,B 0.000,C 90.000,E1 319.299} C_DIS
LIN {X 0.064,Y -485.175,Z 1310.573,A 0.000,B 0.000,C 90.000,E1 319.138} C_DIS
LIN {X 0.171,Y -463.298,Z 1310.560,A 0.000,B 0.000,C 90.000,E1 316.782} C_DIS
LIN {X -0.012,Y -443.766,Z 1310.547,A 0.000,B 0.000,C 90.000,E1 314.433} C_DIS
LIN {X -0.052,Y -425.796,Z 1310.533,A 0.000,B 0.000,C 90.000,E1 311.962} C_DIS
LIN {X 0.054,Y -409.544,Z 1310.519,A 0.000,B 0.000,C 90.000,E1 309.402} C_DIS
LIN {X 0.064,Y -394.887,Z 1310.505,A 0.000,B 0.000,C 90.000,E1 306.790} C_DIS
LIN {X -0.154,Y -389.671,Z 1310.499,A 0.000,B 0.000,C 90.000,E1 305.804} C_DIS
LIN {X -0.191,Y -389.672,Z 1310.499,A 0.000,B 0.000,C 90.000,E1 305.804} C_DIS
LIN {X 0.037,Y -391.347,Z 1310.492,A 0.000,B 0.000,C 90.000,E1 304.485} C_DIS
LIN {X -0.140,Y -397.058,Z 1310.458,A 0.000,B 0.000,C 90.000,E1 298.487} C_DIS
LIN {X 0.165,Y -401.450,Z 1310.427,A 0.000,B 0.000,C 90.000,E1 292.823} C_DIS
LIN {X -0.125,Y -401.677,Z 1310.425,A 0.000,B 0.000,C 90.000,E1 292.514} C_DIS
LIN {X -0.095,Y -404.537,Z 1310.396,A 0.000,B 0.000,C 90.000,E1 287.275} C_DIS
LIN {X 0.005,Y -404.763,Z 1310.394,A 0.000,B 0.000,C 90.000,E1 286.913} C_DIS
LIN {X -0.088,Y -406.150,Z 1310.363,A 0.000,B 0.000,C 90.000,E1 281.366} C_DIS
LIN {X 0.017,Y -405.648,Z 1310.334,A 0.000,B 0.000,C 90.000,E1 276.144} C_DIS
LIN {X 0.021,Y -405.625,Z 1310.332,A 0.000,B 0.000,C 90.000,E1 275.796} C_DIS
LIN {X 0.094,Y -403.554,Z 1310.305,A 0.000,B 0.000,C 90.000,E1 270.917} C_DIS
LIN {X 0.029,Y -403.075,Z 1310.301,A 0.000,B 0.000,C 90.000,E1 270.229} C_DIS
LIN {X -0.144,Y -399.024,Z 1310.272,A 0.000,B 0.000,C 90.000,E1 265.008} C_DIS
LIN {X 0.169,Y -398.149,Z 1310.268,A 0.000,B 0.000,C 90.000,E1 264.261} C_DIS
LIN {X 0.027,Y -392.946,Z 1310.241,A 0.000,B 0.000,C 90.000,E1 259.342} C_DIS
LIN {X -0.015,Y -392.509,Z 1310.239,A 0.000,B 0.000,C 90.000,E1 258.993} C_DIS
LIN {X 0.132,Y -386.143,Z 1310.213,A 0.000,B 0.000,C 90.000,E1 254.338} C_DIS
LIN {X 0.093,Y -385.021,Z 1310.207,A 0.000,B 0.000,C 90.000,E1 253.268} C_DIS
LIN {X -0.034,Y -378.157,Z 1310.183,A 0.000,B 0.000,C 90.000,E1 248.954} C_DIS
LIN {X 0.179,Y -375.917,Z 1310.173,A 0.000,B 0.000,C 90.000,E1 247.102} C_DIS
LIN {X -0.201,Y -369.131,Z 1310.151,A 0.000,B 0.000,C 90.000,E1 243.127} C_DIS
LIN {X 0.028,Y -366.281,Z 1310.138,A 0.000,B 0.000,C 90.000,E1 240.873} C_DIS
LIN {X -0.002,Y -365.045,Z 1310.135,A 0.000,B 0.000,C 90.000,E1 240.205} C_DIS
LIN {X -0.040,Y -365.050,Z 1310.135,A 0.000,B 0.000,C 90.000,E1 240.205} C_DIS
LIN {X -0.054,Y -376.507,Z 1310.119,A 0.000,B 0.000,C 90.000,E1 237.375} C_DIS
LIN {X 0.074,Y -389.097,Z 1310.104,A 0.000,B 0.000,C 90.000,E1 234.642} C_DIS
LIN {X 0.104,Y -403.152,Z 1310.089,A 0.000,B 0.000,C 90.000,E1 231.984} C_DIS
LIN {X 0.206,Y -418.776,Z 1310.075,A 0.000,B 0.000,C 90.000,E1 229.380} C_DIS
LIN {X -0.155,Y -436.080,Z 1310.061,A 0.000,B 0.000,C 90.000,E1 226.905} C_DIS
LIN {X 0.010,Y -444.768,Z 1310.054,A 0.000,B 0.000,C 90.000,E1 225.729} C_DIS
LIN {X -0.001,Y -445.877,Z 1310.053,A 0.000,B 0.000,C 90.000,E1 225.567} C_DIS
LIN {X -0.011,Y -446.609,Z 1310.052,A 0.000,B 0.000,C 90.000,E1 225.405} C_DIS
LIN {X -0.023,Y -447.612,Z 1310.051,A 0.000,B 0.000,C 90.000,E1 225.081} C_DIS
LIN {X -0.032,Y -448.325,Z 1310.049,A 0.000,B 0.000,C 90.000,E1 224.757} C_DIS
LIN {X -0.040,Y -449.296,Z 1310.045,A 0.000,B 0.000,C 90.000,E1 224.109} C_DIS
LIN {X -0.040,Y -449.902,Z 1310.042,A 0.000,B 0.000,C 90.000,E1 223.461} C_DIS
LIN {X -0.010,Y -450.429,Z 1310.036,A 0.000,B 0.000,C 90.000,E1 222.486} C_DIS
LIN {X -0.001,Y -450.643,Z 1310.031,A 0.000,B 0.000,C 90.000,E1 221.515} C_DIS
LIN {X -0.078,Y -452.229,Z 1310.011,A 0.000,B 0.000,C 90.000,E1 217.971} C_DIS
LIN {X -0.224,Y -453.515,Z 1310.002,A 0.000,B 0.000,C 90.000,E1 216.377} C_DIS
LIN {X 0.108,Y -455.190,Z 1309.991,A 0.000,B 0.000,C 90.000,E1 214.405} C_DIS
LIN {X 0.082,Y -457.472,Z 1309.979,A 0.000,B 0.000,C 90.000,E1 212.163} C_DIS
LIN {X -0.150,Y -461.246,Z 1309.961,A 0.000,B 0.000,C 90.000,E1 208.999} C_DIS
LIN {X 0.021,Y -464.762,Z 1309.947,A 0.000,B 0.000,C 90.000,E1 206.437} C_DIS
LIN {X 0.110,Y -468.457,Z 1309.933,A 0.000,B 0.000,C 90.000,E1 203.898} C_DIS
LIN {X -0.036,Y -471.478,Z 1309.921,A 0.000,B 0.000,C 90.000,E1 201.716} C_DIS
LIN {X 0.183,Y -474.148,Z 1309.910,A 0.000,B 0.000,C 90.000,E1 199.812} C_DIS
LIN {X 0.122,Y -477.362,Z 1309.898,A 0.000,B 0.000,C 90.000,E1 197.638} C_DIS
LIN {X -0.152,Y -481.027,Z 1309.884,A 0.000,B 0.000,C 90.000,E1 195.190} C_DIS
LIN {X 0.173,Y -483.658,Z 1309.874,A 0.000,B 0.000,C 90.000,E1 193.300} C_DIS
LIN {X -0.027,Y -486.304,Z 1309.864,A 0.000,B 0.000,C 90.000,E1 191.478} C_DIS
LIN {X 0.211,Y -488.873,Z 1309.854,A 0.000,B 0.000,C 90.000,E1 189.613} C_DIS
LIN {X -0.063,Y -491.421,Z 1309.843,A 0.000,B 0.000,C 90.000,E1 187.814} C_DIS
LIN {X 0.244,Y -493.496,Z 1309.835,A 0.000,B 0.000,C 90.000,E1 186.258} C_DIS
LIN {X 0.097,Y -495.452,Z 1309.827,A 0.000,B 0.000,C 90.000,E1 184.759} C_DIS
LIN {X 0.046,Y -496.864,Z 1309.820,A 0.000,B 0.000,C 90.000,E1 183.555} C_DIS
LIN {X 0.157,Y -497.858,Z 1309.815,A 0.000,B 0.000,C 90.000,E1 182.636} C_DIS
LIN {X 0.015,Y -499.295,Z 1309.806,A 0.000,B 0.000,C 90.000,E1 181.146} C_DIS
LIN {X 0.012,Y -500.298,Z 1309.800,A 0.000,B 0.000,C 90.000,E1 179.943} C_DIS
LIN {X -0.098,Y -501.194,Z 1309.791,A 0.000,B 0.000,C 90.000,E1 178.453} C_DIS
LIN {X 0.058,Y -501.611,Z 1309.786,A 0.000,B 0.000,C 90.000,E1 177.535} C_DIS
LIN {X -0.021,Y -501.901,Z 1309.778,A 0.000,B 0.000,C 90.000,E1 176.045} C_DIS
LIN {X 0.185,Y -501.869,Z 1309.773,A 0.000,B 0.000,C 90.000,E1 175.122} C_DIS
LIN {X -0.149,Y -501.633,Z 1309.768,A 0.000,B 0.000,C 90.000,E1 174.261} C_DIS
LIN {X -0.150,Y -500.963,Z 1309.760,A 0.000,B 0.000,C 90.000,E1 172.761} C_DIS
LIN {X -0.023,Y -499.917,Z 1309.753,A 0.000,B 0.000,C 90.000,E1 171.546} C_DIS
LIN {X 0.163,Y -498.797,Z 1309.748,A 0.000,B 0.000,C 90.000,E1 170.622} C_DIS
LIN {X -0.073,Y -497.349,Z 1309.743,A 0.000,B 0.000,C 90.000,E1 169.746} C_DIS
LIN {X 0.164,Y -495.722,Z 1309.738,A 0.000,B 0.000,C 90.000,E1 168.814} C_DIS
LIN {X 0.187,Y -492.224,Z 1309.730,A 0.000,B 0.000,C 90.000,E1 167.297} C_DIS
LIN {X -0.011,Y -489.652,Z 1309.724,A 0.000,B 0.000,C 90.000,E1 166.408} C_DIS
LIN {X -0.115,Y -487.898,Z 1309.721,A 0.000,B 0.000,C 90.000,E1 165.811} C_DIS
LIN {X -0.009,Y -483.612,Z 1309.714,A 0.000,B 0.000,C 90.000,E1 164.574} C_DIS
LIN {X -0.079,Y -479.014,Z 1309.708,A 0.000,B 0.000,C 90.000,E1 163.504} C_DIS
LIN {X 0.151,Y -469.787,Z 1309.699,A 0.000,B 0.000,C 90.000,E1 161.764} C_DIS
LIN {X 0.052,Y -466.573,Z 1309.695,A 0.000,B 0.000,C 90.000,E1 161.148} C_DIS
LIN {X -0.219,Y -463.995,Z 1309.692,A 0.000,B 0.000,C 90.000,E1 160.550} C_DIS
LIN {X 0.085,Y -461.970,Z 1309.688,A 0.000,B 0.000,C 90.000,E1 159.880} C_DIS
LIN {X -0.061,Y -460.618,Z 1309.685,A 0.000,B 0.000,C 90.000,E1 159.263} C_DIS
LIN {X 0.116,Y -460.325,Z 1309.684,A 0.000,B 0.000,C 90.000,E1 159.082} C_DIS
LIN {X -0.138,Y -460.316,Z 1309.683,A 0.000,B 0.000,C 90.000,E1 158.954} C_DIS
LIN {X -0.179,Y -460.801,Z 1309.679,A 0.000,B 0.000,C 90.000,E1 158.284} C_DIS
LIN {X 0.207,Y -461.007,Z 1309.679,A 0.000,B 0.000,C 90.000,E1 158.156} C_DIS
LIN {X -0.107,Y -461.975,Z 1309.678,A 0.000,B 0.000,C 90.000,E1 158.028} C_DIS
LIN {X 0.054,Y -464.506,Z 1309.676,A 0.000,B 0.000,C 90.000,E1 157.741} C_DIS
LIN {X 0.199,Y -465.920,Z 1309.675,A 0.000,B 0.000,C 90.000,E1 157.539} C_DIS
LIN {X 0.027,Y -469.096,Z 1309.674,A 0.000,B 0.000,C 90.000,E1 157.283} C_DIS
LIN {X -0.275,Y -472.216,Z 1309.672,A 0.000,B 0.000,C 90.000,E1 157.050} C_DIS
LIN {X 0.070,Y -484.967,Z 1309.667,A 0.000,B 0.000,C 90.000,E1 155.973} C_DIS
LIN {X -0.038,Y -490.869,Z 1309.664,A 0.000,B 0.000,C 90.000,E1 155.485} C_DIS
LIN {X -0.046,Y -495.187,Z 1309.662,A 0.000,B 0.000,C 90.000,E1 155.101} C_DIS
LIN {X -0.036,Y -501.875,Z 1309.658,A 0.000,B 0.000,C 90.000,E1 154.460} C_DIS
LIN {X 0.220,Y -505.941,Z 1309.656,A 0.000,B 0.000,C 90.000,E1 154.024} C_DIS
LIN {X -0.265,Y -511.158,Z 1309.653,A 0.000,B 0.000,C 90.000,E1 153.512} C_DIS
LIN {X -0.068,Y -515.024,Z 1309.650,A 0.000,B 0.000,C 90.000,E1 153.050} C_DIS
LIN {X -0.275,Y -519.717,Z 1309.647,A 0.000,B 0.000,C 90.000,E1 152.487} C_DIS
LIN {X -0.233,Y -523.910,Z 1309.644,A 0.000,B 0.000,C 90.000,E1 151.897} C_DIS
LIN {X -0.156,Y -527.597,Z 1309.641,A 0.000,B 0.000,C 90.000,E1 151.307} C_DIS
LIN {X -0.202,Y -531.315,Z 1309.637,A 0.000,B 0.000,C 90.000,E1 150.589} C_DIS
LIN {X -0.069,Y -533.781,Z 1309.633,A 0.000,B 0.000,C 90.000,E1 149.999} C_DIS
LIN {X 0.065,Y -536.602,Z 1309.629,A 0.000,B 0.000,C 90.000,E1 149.125} C_DIS
LIN {X 0.232,Y -538.149,Z 1309.625,A 0.000,B 0.000,C 90.000,E1 148.535} C_DIS
LIN {X -0.044,Y -540.015,Z 1309.621,A 0.000,B 0.000,C 90.000,E1 147.709} C_DIS
LIN {X 0.143,Y -541.099,Z 1309.617,A 0.000,B 0.000,C 90.000,E1 147.120} C_DIS
LIN {X -0.102,Y -542.349,Z 1309.613,A 0.000,B 0.000,C 90.000,E1 146.294} C_DIS
LIN {X -0.133,Y -544.122,Z 1309.606,A 0.000,B 0.000,C 90.000,E1 145.022} C_DIS
LIN {X 0.113,Y -544.892,Z 1309.604,A 0.000,B 0.000,C 90.000,E1 144.609} C_DIS
LIN {X 0.071,Y -544.921,Z 1309.604,A 0.000,B 0.000,C 90.000,E1 144.609} C_DIS
LIN {X 0.033,Y -545.529,Z 1309.603,A 0.000,B 0.000,C 90.000,E1 144.529} C_DIS
LIN {X -0.108,Y -546.289,Z 1309.602,A 0.000,B 0.000,C 90.000,E1 144.402} C_DIS
LIN {X -0.116,Y -546.884,Z 1309.601,A 0.000,B 0.000,C 90.000,E1 144.196} C_DIS
LIN {X -0.158,Y -546.959,Z 1309.601,A 0.000,B 0.000,C 90.000,E1 144.196} C_DIS
LIN {X 0.375,Y -551.861,Z 1309.600,A 0.000,B 0.000,C 90.000,E1 143.909} C_DIS
LIN {X 0.016,Y -562.118,Z 1309.598,A 0.000,B 0.000,C 90.000,E1 143.543} C_DIS
LIN {X -0.117,Y -565.507,Z 1309.597,A 0.000,B 0.000,C 90.000,E1 143.417} C_DIS
LIN {X -0.288,Y -571.516,Z 1309.595,A 0.000,B 0.000,C 90.000,E1 143.130} C_DIS
LIN {X -0.181,Y -577.605,Z 1309.593,A 0.000,B 0.000,C 90.000,E1 142.763} C_DIS
LIN {X -0.171,Y -582.034,Z 1309.592,A 0.000,B 0.000,C 90.000,E1 142.477} C_DIS
LIN {X 0.083,Y -587.695,Z 1309.589,A 0.000,B 0.000,C 90.000,E1 142.029} C_DIS
LIN {X -0.044,Y -593.056,Z 1309.587,A 0.000,B 0.000,C 90.000,E1 141.582} C_DIS
LIN {X -0.364,Y -596.947,Z 1309.585,A 0.000,B 0.000,C 90.000,E1 141.251} C_DIS
LIN {X 0.111,Y -601.646,Z 1309.582,A 0.000,B 0.000,C 90.000,E1 140.723} C_DIS
LIN {X 0.246,Y -606.147,Z 1309.579,A 0.000,B 0.000,C 90.000,E1 140.194} C_DIS
LIN {X 0.042,Y -609.324,Z 1309.577,A 0.000,B 0.000,C 90.000,E1 139.828} C_DIS
LIN {X -0.161,Y -614.049,Z 1309.573,A 0.000,B 0.000,C 90.000,E1 139.218} C_DIS
LIN {X -0.393,Y -616.918,Z 1309.571,A 0.000,B 0.000,C 90.000,E1 138.852} C_DIS
LIN {X 0.101,Y -621.209,Z 1309.568,A 0.000,B 0.000,C 90.000,E1 138.162} C_DIS
LIN {X 0.267,Y -624.312,Z 1309.565,A 0.000,B 0.000,C 90.000,E1 137.634} C_DIS
LIN {X 0.010,Y -628.823,Z 1309.561,A 0.000,B 0.000,C 90.000,E1 136.905} C_DIS
LIN {X -0.161,Y -631.054,Z 1309.558,A 0.000,B 0.000,C 90.000,E1 136.539} C_DIS
LIN {X 0.003,Y -634.488,Z 1309.555,A 0.000,B 0.000,C 90.000,E1 135.891} C_DIS
LIN {X -0.204,Y -637.200,Z 1309.552,A 0.000,B 0.000,C 90.000,E1 135.405} C_DIS
LIN {X 0.175,Y -639.249,Z 1309.550,A 0.000,B 0.000,C 90.000,E1 135.000} C_DIS
LIN {X 0.334,Y -643.807,Z 1309.545,A 0.000,B 0.000,C 90.000,E1 134.109} C_DIS
LIN {X 0.041,Y -649.472,Z 1309.539,A 0.000,B 0.000,C 90.000,E1 133.014} C_DIS
LIN {X -0.079,Y -652.597,Z 1309.536,A 0.000,B 0.000,C 90.000,E1 132.405} C_DIS
LIN {X 0.232,Y -657.545,Z 1309.530,A 0.000,B 0.000,C 90.000,E1 131.391} C_DIS
LIN {X -0.332,Y -662.219,Z 1309.525,A 0.000,B 0.000,C 90.000,E1 130.458} C_DIS
LIN {X -0.322,Y -665.555,Z 1309.521,A 0.000,B 0.000,C 90.000,E1 129.725} C_DIS
LIN {X -0.290,Y -669.730,Z 1309.515,A 0.000,B 0.000,C 90.000,E1 128.749} C_DIS
LIN {X 0.319,Y -673.521,Z 1309.510,A 0.000,B 0.000,C 90.000,E1 127.729} C_DIS
LIN {X 0.034,Y -677.018,Z 1309.504,A 0.000,B 0.000,C 90.000,E1 126.790} C_DIS
LIN {X -0.219,Y -679.413,Z 1309.500,A 0.000,B 0.000,C 90.000,E1 126.091} C_DIS
LIN {X 0.117,Y -682.226,Z 1309.495,A 0.000,B 0.000,C 90.000,E1 125.105} C_DIS
LIN {X 0.300,Y -683.604,Z 1309.492,A 0.000,B 0.000,C 90.000,E1 124.612} C_DIS
LIN {X -0.266,Y -685.974,Z 1309.487,A 0.000,B 0.000,C 90.000,E1 123.706} C_DIS
LIN {X -0.231,Y -688.058,Z 1309.482,A 0.000,B 0.000,C 90.000,E1 122.752} C_DIS
LIN {X 0.197,Y -689.426,Z 1309.478,A 0.000,B 0.000,C 90.000,E1 122.005} C_DIS
LIN {X -0.085,Y -691.046,Z 1309.473,A 0.000,B 0.000,C 90.000,E1 121.082} C_DIS
LIN {X 0.248,Y -692.775,Z 1309.466,A 0.000,B 0.000,C 90.000,E1 119.873} C_DIS
LIN {X -0.233,Y -693.623,Z 1309.462,A 0.000,B 0.000,C 90.000,E1 119.205} C_DIS
LIN {X -0.103,Y -694.388,Z 1309.458,A 0.000,B 0.000,C 90.000,E1 118.487} C_DIS
LIN {X 0.034,Y -694.829,Z 1309.454,A 0.000,B 0.000,C 90.000,E1 117.769} C_DIS
LIN {X -0.256,Y -695.212,Z 1309.448,A 0.000,B 0.000,C 90.000,E1 116.616} C_DIS
LIN {X -0.117,Y -695.080,Z 1309.444,A 0.000,B 0.000,C 90.000,E1 115.899} C_DIS
LIN {X 0.088,Y -694.850,Z 1309.441,A 0.000,B 0.000,C 90.000,E1 115.412} C_DIS
LIN {X -0.037,Y -694.369,Z 1309.439,A 0.000,B 0.000,C 90.000,E1 114.951} C_DIS
LIN {X 0.173,Y -693.624,Z 1309.436,A 0.000,B 0.000,C 90.000,E1 114.463} C_DIS
LIN {X -0.212,Y -693.035,Z 1309.435,A 0.000,B 0.000,C 90.000,E1 114.259} C_DIS
LIN {X -0.005,Y -691.520,Z 1309.432,A 0.000,B 0.000,C 90.000,E1 113.770} C_DIS
LIN {X -0.323,Y -688.119,Z 1309.429,A 0.000,B 0.000,C 90.000,E1 113.206} C_DIS
LIN {X -0.209,Y -687.062,Z 1309.428,A 0.000,B 0.000,C 90.000,E1 113.078} C_DIS
LIN {X -0.329,Y -681.467,Z 1309.426,A 0.000,B 0.000,C 90.000,E1 112.642} C_DIS
LIN {X -0.096,Y -679.627,Z 1309.425,A 0.000,B 0.000,C 90.000,E1 112.514} C_DIS
LIN {X -0.118,Y -673.194,Z 1309.424,A 0.000,B 0.000,C 90.000,E1 112.280} C_DIS
LIN {X -0.042,Y -667.749,Z 1309.423,A 0.000,B 0.000,C 90.000,E1 112.153} C_DIS
LIN {X 0.042,Y -663.830,Z 1309.423,A 0.000,B 0.000,C 90.000,E1 112.078} C_DIS
LIN {X -0.241,Y -655.117,Z 1309.422,A 0.000,B 0.000,C 90.000,E1 112.025} C_DIS
LIN {X 0.155,Y -650.009,Z 1309.422,A 0.000,B 0.000,C 90.000,E1 111.972} C_DIS
LIN {X 0.385,Y -645.214,Z 1309.422,A 0.000,B 0.000,C 90.000,E1 111.897} C_DIS
LIN {X 0.142,Y -643.949,Z 1309.422,A 0.000,B 0.000,C 90.000,E1 111.897} C_DIS
LIN {X 0.005,Y -642.027,Z 1309.421,A 0.000,B 0.000,C 90.000,E1 111.844} C_DIS
LIN {X -0.036,Y -641.933,Z 1309.421,A 0.000,B 0.000,C 90.000,E1 111.844} C_DIS
LIN {X -0.187,Y -642.820,Z 1309.420,A 0.000,B 0.000,C 90.000,E1 111.663} C_DIS
LIN {X -0.159,Y -643.573,Z 1309.420,A 0.000,B 0.000,C 90.000,E1 111.535} C_DIS
LIN {X -0.165,Y -651.368,Z 1309.414,A 0.000,B 0.000,C 90.000,E1 110.536} C_DIS
LIN {X 0.207,Y -655.605,Z 1309.411,A 0.000,B 0.000,C 90.000,E1 109.885} C_DIS
LIN {X 0.228,Y -659.235,Z 1309.407,A 0.000,B 0.000,C 90.000,E1 109.268} C_DIS
LIN {X 0.059,Y -662.405,Z 1309.404,A 0.000,B 0.000,C 90.000,E1 108.671} C_DIS
LIN {X -0.027,Y -665.691,Z 1309.400,A 0.000,B 0.000,C 90.000,E1 107.946} C_DIS
LIN {X -0.085,Y -668.573,Z 1309.396,A 0.000,B 0.000,C 90.000,E1 107.221} C_DIS
LIN {X -0.046,Y -670.254,Z 1309.393,A 0.000,B 0.000,C 90.000,E1 106.732} C_DIS
LIN {X -0.257,Y -672.435,Z 1309.389,A 0.000,B 0.000,C 90.000,E1 106.024} C_DIS
LIN {X -0.263,Y -674.232,Z 1309.385,A 0.000,B 0.000,C 90.000,E1 105.300} C_DIS
LIN {X 0.221,Y -675.740,Z 1309.381,A 0.000,B 0.000,C 90.000,E1 104.537} C_DIS
LIN {X 0.071,Y -677.021,Z 1309.377,A 0.000,B 0.000,C 90.000,E1 103.828} C_DIS
LIN {X -0.068,Y -677.848,Z 1309.373,A 0.000,B 0.000,C 90.000,E1 103.119} C_DIS
LIN {X -0.158,Y -678.217,Z 1309.370,A 0.000,B 0.000,C 90.000,E1 102.647} C_DIS
LIN {X 0.231,Y -678.487,Z 1309.366,A 0.000,B 0.000,C 90.000,E1 101.895} C_DIS
LIN {X 0.146,Y -678.443,Z 1309.364,A 0.000,B 0.000,C 90.000,E1 101.422} C_DIS
LIN {X 0.008,Y -677.944,Z 1309.360,A 0.000,B 0.000,C 90.000,E1 100.715} C_DIS
LIN {X -0.213,Y -677.436,Z 1309.357,A 0.000,B 0.000,C 90.000,E1 100.254} C_DIS
LIN {X 0.350,Y -676.674,Z 1309.354,A 0.000,B 0.000,C 90.000,E1 99.726} C_DIS
LIN {X 0.127,Y -675.614,Z 1309.352,A 0.000,B 0.000,C 90.000,E1 99.265} C_DIS
LIN {X -0.099,Y -674.207,Z 1309.349,A 0.000,B 0.000,C 90.000,E1 98.803} C_DIS
LIN {X 0.265,Y -671.462,Z 1309.345,A 0.000,B 0.000,C 90.000,E1 98.049} C_DIS
LIN {X 0.017,Y -669.281,Z 1309.342,A 0.000,B 0.000,C 90.000,E1 97.587} C_DIS
LIN {X -0.247,Y -666.165,Z 1309.339,A 0.000,B 0.000,C 90.000,E1 97.004} C_DIS
LIN {X 0.036,Y -662.823,Z 1309.335,A 0.000,B 0.000,C 90.000,E1 96.372} C_DIS
LIN {X -0.268,Y -659.916,Z 1309.333,A 0.000,B 0.000,C 90.000,E1 95.910} C_DIS
LIN {X 0.064,Y -656.670,Z 1309.330,A 0.000,B 0.000,C 90.000,E1 95.391} C_DIS
LIN {X -0.337,Y -653.251,Z 1309.327,A 0.000,B 0.000,C 90.000,E1 94.935} C_DIS
LIN {X -0.051,Y -649.476,Z 1309.325,A 0.000,B 0.000,C 90.000,E1 94.416} C_DIS
LIN {X 0.127,Y -644.317,Z 1309.321,A 0.000,B 0.000,C 90.000,E1 93.784} C_DIS
LIN {X 0.185,Y -636.578,Z 1309.316,A 0.000,B 0.000,C 90.000,E1 92.922} C_DIS
LIN {X 0.066,Y -629.401,Z 1309.312,A 0.000,B 0.000,C 90.000,E1 92.178} C_DIS
LIN {X 0.315,Y -624.416,Z 1309.309,A 0.000,B 0.000,C 90.000,E1 91.661} C_DIS
LIN {X 0.021,Y -616.249,Z 1309.305,A 0.000,B 0.000,C 90.000,E1 90.974} C_DIS
LIN {X -0.264,Y -608.666,Z 1309.302,A 0.000,B 0.000,C 90.000,E1 90.458} C_DIS
LIN {X -0.127,Y -602.281,Z 1309.300,A 0.000,B 0.000,C 90.000,E1 90.057} C_DIS
LIN {X -0.191,Y -595.659,Z 1309.298,A 0.000,B 0.000,C 90.000,E1 89.714} C_DIS
LIN {X 0.168,Y -588.649,Z 1309.297,A 0.000,B 0.000,C 90.000,E1 89.370} C_DIS
LIN {X 0.182,Y -576.452,Z 1309.294,A 0.000,B 0.000,C 90.000,E1 88.912} C_DIS
LIN {X 0.041,Y -572.483,Z 1309.293,A 0.000,B 0.000,C 90.000,E1 88.740} C_DIS
LIN {X -0.003,Y -572.440,Z 1309.293,A 0.000,B 0.000,C 90.000,E1 88.740} C_DIS
LIN {X 0.092,Y -570.666,Z 1309.292,A 0.000,B 0.000,C 90.000,E1 88.511} C_DIS
LIN {X 0.050,Y -570.653,Z 1309.292,A 0.000,B 0.000,C 90.000,E1 88.511} C_DIS
LIN {X -0.005,Y -570.397,Z 1309.291,A 0.000,B 0.000,C 90.000,E1 88.282} C_DIS
LIN {X 0.166,Y -570.592,Z 1309.287,A 0.000,B 0.000,C 90.000,E1 87.650} C_DIS
LIN {X 0.275,Y -571.879,Z 1309.280,A 0.000,B 0.000,C 90.000,E1 86.274} C_DIS
LIN {X -0.066,Y -574.507,Z 1309.266,A 0.000,B 0.000,C 90.000,E1 83.856} C_DIS
LIN {X -0.265,Y -577.363,Z 1309.252,A 0.000,B 0.000,C 90.000,E1 81.432} C_DIS
LIN {X -0.206,Y -579.302,Z 1309.243,A 0.000,B 0.000,C 90.000,E1 79.803} C_DIS
LIN {X 0.234,Y -580.755,Z 1309.236,A 0.000,B 0.000,C 90.000,E1 78.409} C_DIS
LIN {X 0.238,Y -582.005,Z 1309.228,A 0.000,B 0.000,C 90.000,E1 77.061} C_DIS
LIN {X 0.168,Y -582.913,Z 1309.222,A 0.000,B 0.000,C 90.000,E1 75.992} C_DIS
LIN {X -0.210,Y -583.890,Z 1309.215,A 0.000,B 0.000,C 90.000,E1 74.685} C_DIS
LIN {X -0.012,Y -584.787,Z 1309.207,A 0.000,B 0.000,C 90.000,E1 73.323} C_DIS
LIN {X -0.198,Y -585.645,Z 1309.200,A 0.000,B 0.000,C 90.000,E1 72.000} C_DIS
LIN {X 0.042,Y -586.674,Z 1309.191,A 0.000,B 0.000,C 90.000,E1 70.369} C_DIS
LIN {X -0.174,Y -587.913,Z 1309.181,A 0.000,B 0.000,C 90.000,E1 68.518} C_DIS
LIN {X -0.240,Y -588.994,Z 1309.172,A 0.000,B 0.000,C 90.000,E1 66.922} C_DIS
LIN {X -0.179,Y -590.259,Z 1309.161,A 0.000,B 0.000,C 90.000,E1 65.049} C_DIS
LIN {X -0.114,Y -591.548,Z 1309.151,A 0.000,B 0.000,C 90.000,E1 63.179} C_DIS
LIN {X -0.201,Y -593.652,Z 1309.138,A 0.000,B 0.000,C 90.000,E1 60.795} C_DIS
LIN {X -0.076,Y -595.753,Z 1309.126,A 0.000,B 0.000,C 90.000,E1 58.663} C_DIS
LIN {X -0.309,Y -597.728,Z 1309.116,A 0.000,B 0.000,C 90.000,E1 56.834} C_DIS
LIN {X -0.069,Y -599.431,Z 1309.107,A 0.000,B 0.000,C 90.000,E1 55.229} C_DIS
LIN {X 0.208,Y -600.888,Z 1309.098,A 0.000,B 0.000,C 90.000,E1 53.623} C_DIS
LIN {X -0.234,Y -602.040,Z 1309.091,A 0.000,B 0.000,C 90.000,E1 52.351} C_DIS
LIN {X 0.297,Y -602.863,Z 1309.085,A 0.000,B 0.000,C 90.000,E1 51.251} C_DIS
LIN {X 0.032,Y -603.972,Z 1309.076,A 0.000,B 0.000,C 90.000,E1 49.703} C_DIS
LIN {X -0.128,Y -604.468,Z 1309.072,A 0.000,B 0.000,C 90.000,E1 48.933} C_DIS
LIN {X -0.029,Y -604.786,Z 1309.066,A 0.000,B 0.000,C 90.000,E1 47.877} C_DIS
LIN {X 0.082,Y -605.007,Z 1309.057,A 0.000,B 0.000,C 90.000,E1 46.296} C_DIS
LIN {X -0.036,Y -605.066,Z 1309.050,A 0.000,B 0.000,C 90.000,E1 45.000} C_DIS
LIN {X 0.041,Y -604.910,Z 1309.044,A 0.000,B 0.000,C 90.000,E1 43.947} C_DIS
LIN {X 0.155,Y -604.493,Z 1309.036,A 0.000,B 0.000,C 90.000,E1 42.366} C_DIS
LIN {X 0.052,Y -604.045,Z 1309.028,A 0.000,B 0.000,C 90.000,E1 41.067} C_DIS
LIN {X 0.146,Y -603.554,Z 1309.022,A 0.000,B 0.000,C 90.000,E1 40.011} C_DIS
LIN {X -0.150,Y -603.078,Z 1309.017,A 0.000,B 0.000,C 90.000,E1 38.991} C_DIS
LIN {X 0.144,Y -602.584,Z 1309.012,A 0.000,B 0.000,C 90.000,E1 38.177} C_DIS
LIN {X -0.164,Y -601.674,Z 1309.006,A 0.000,B 0.000,C 90.000,E1 37.156} C_DIS
LIN {X -0.004,Y -600.497,Z 1309.001,A 0.000,B 0.000,C 90.000,E1 36.091} C_DIS
LIN {X 0.034,Y -598.590,Z 1308.993,A 0.000,B 0.000,C 90.000,E1 34.771} C_DIS
LIN {X 0.143,Y -596.745,Z 1308.987,A 0.000,B 0.000,C 90.000,E1 33.706} C_DIS
LIN {X -0.332,Y -595.084,Z 1308.983,A 0.000,B 0.000,C 90.000,E1 32.959} C_DIS
LIN {X -0.108,Y -592.487,Z 1308.977,A 0.000,B 0.000,C 90.000,E1 31.878} C_DIS
LIN {X 0.189,Y -590.211,Z 1308.973,A 0.000,B 0.000,C 90.000,E1 31.052} C_DIS
LIN {X 0.151,Y -587.605,Z 1308.968,A 0.000,B 0.000,C 90.000,E1 30.256} C_DIS
LIN {X 0.088,Y -584.600,Z 1308.964,A 0.000,B 0.000,C 90.000,E1 29.461} C_DIS
LIN {X -0.161,Y -582.328,Z 1308.961,A 0.000,B 0.000,C 90.000,E1 28.949} C_DIS
LIN {X 0.230,Y -578.627,Z 1308.956,A 0.000,B 0.000,C 90.000,E1 28.103} C_DIS
LIN {X -0.018,Y -573.690,Z 1308.951,A 0.000,B 0.000,C 90.000,E1 27.180} C_DIS
LIN {X 0.009,Y -569.025,Z 1308.947,A 0.000,B 0.000,C 90.000,E1 26.360} C_DIS
LIN {X 0.083,Y -564.724,Z 1308.943,A 0.000,B 0.000,C 90.000,E1 25.668} C_DIS
LIN {X -0.289,Y -561.052,Z 1308.940,A 0.000,B 0.000,C 90.000,E1 25.155} C_DIS
LIN {X -0.078,Y -558.141,Z 1308.937,A 0.000,B 0.000,C 90.000,E1 24.719} C_DIS
LIN {X 0.012,Y -553.952,Z 1308.934,A 0.000,B 0.000,C 90.000,E1 24.155} C_DIS
LIN {X -0.043,Y -548.375,Z 1308.930,A 0.000,B 0.000,C 90.000,E1 23.462} C_DIS
LIN {X 0.099,Y -544.886,Z 1308.928,A 0.000,B 0.000,C 90.000,E1 23.025} C_DIS
LIN {X -0.118,Y -537.600,Z 1308.923,A 0.000,B 0.000,C 90.000,E1 22.206} C_DIS
LIN {X -0.117,Y -532.554,Z 1308.920,A 0.000,B 0.000,C 90.000,E1 21.642} C_DIS
LIN {X -0.086,Y -522.201,Z 1308.914,A 0.000,B 0.000,C 90.000,E1 20.536} C_DIS
LIN {X -0.205,Y -512.953,Z 1308.909,A 0.000,B 0.000,C 90.000,E1 19.577} C_DIS
LIN {X 0.255,Y -501.938,Z 1308.903,A 0.000,B 0.000,C 90.000,E1 18.417} C_DIS
LIN {X -0.266,Y -490.888,Z 1308.897,A 0.000,B 0.000,C 90.000,E1 17.402} C_DIS
LIN {X 0.011,Y -483.670,Z 1308.893,A 0.000,B 0.000,C 90.000,E1 16.677} C_DIS
LIN {X 0.144,Y -473.562,Z 1308.888,A 0.000,B 0.000,C 90.000,E1 15.733} C_DIS
LIN {X -0.143,Y -456.038,Z 1308.879,A 0.000,B 0.000,C 90.000,E1 14.175} C_DIS
LIN {X -0.191,Y -434.258,Z 1308.867,A 0.000,B 0.000,C 90.000,E1 12.063} C_DIS
LIN {X -0.116,Y -419.940,Z 1308.859,A 0.000,B 0.000,C 90.000,E1 10.546} C_DIS
LIN {X 0.070,Y -408.475,Z 1308.852,A 0.000,B 0.000,C 90.000,E1 9.265} C_DIS
LIN {X 0.005,Y -398.673,Z 1308.845,A 0.000,B 0.000,C 90.000,E1 8.163} C_DIS
LIN {X 0.032,Y -397.436,Z 1308.844,A 0.000,B 0.000,C 90.000,E1 7.992} C_DIS
LIN {X 0.112,Y -395.380,Z 1308.843,A 0.000,B 0.000,C 90.000,E1 7.644} C_DIS
LIN {X 0.074,Y -395.402,Z 1308.843,A 0.000,B 0.000,C 90.000,E1 7.644} C_DIS
LIN {X -0.052,Y -396.198,Z 1308.842,A 0.000,B 0.000,C 90.000,E1 7.530} C_DIS
LIN {X 0.113,Y -399.800,Z 1308.840,A 0.000,B 0.000,C 90.000,E1 7.182} C_DIS
LIN {X -0.135,Y -415.683,Z 1308.834,A 0.000,B 0.000,C 90.000,E1 6.201} C_DIS
LIN {X -0.005,Y -423.698,Z 1308.831,A 0.000,B 0.000,C 90.000,E1 5.625} C_DIS
LIN {X 0.169,Y -432.941,Z 1308.827,A 0.000,B 0.000,C 90.000,E1 4.878} C_DIS
LIN {X -0.075,Y -437.532,Z 1308.825,A 0.000,B 0.000,C 90.000,E1 4.531} C_DIS
LIN {X -0.124,Y -443.546,Z 1308.822,A 0.000,B 0.000,C 90.000,E1 4.012} C_DIS
LIN {X 0.103,Y -449.436,Z 1308.819,A 0.000,B 0.000,C 90.000,E1 3.440} C_DIS
LIN {X -0.184,Y -455.231,Z 1308.816,A 0.000,B 0.000,C 90.000,E1 2.922} C_DIS
LIN {X -0.144,Y -460.892,Z 1308.813,A 0.000,B 0.000,C 90.000,E1 2.350} C_DIS
LIN {X -0.072,Y -467.638,Z 1308.809,A 0.000,B 0.000,C 90.000,E1 1.604} C_DIS
LIN {X 0.011,Y -472.914,Z 1308.805,A 0.000,B 0.000,C 90.000,E1 0.974} C_DIS
LIN {X 0.204,Y -478.883,Z 1308.801,A 0.000,B 0.000,C 90.000,E1 0.172} C_DIS
LIN {X 0.142,Y -484.996,Z 1308.796,A 0.000,B 0.000,C 90.000,E1 359.312} C_DIS
LIN {X -0.052,Y -489.981,Z 1308.792,A 0.000,B 0.000,C 90.000,E1 358.568} C_DIS
LIN {X -0.187,Y -494.587,Z 1308.788,A 0.000,B 0.000,C 90.000,E1 357.822} C_DIS
LIN {X 0.019,Y -498.124,Z 1308.784,A 0.000,B 0.000,C 90.000,E1 357.192} C_DIS
LIN {X 0.154,Y -502.892,Z 1308.779,A 0.000,B 0.000,C 90.000,E1 356.274} C_DIS
LIN {X 0.145,Y -506.615,Z 1308.775,A 0.000,B 0.000,C 90.000,E1 355.527} C_DIS
LIN {X 0.172,Y -510.102,Z 1308.771,A 0.000,B 0.000,C 90.000,E1 354.780} C_DIS
LIN {X 0.190,Y -514.671,Z 1308.765,A 0.000,B 0.000,C 90.000,E1 353.742} C_DIS
LIN {X 0.069,Y -517.079,Z 1308.762,A 0.000,B 0.000,C 90.000,E1 353.166} C_DIS
LIN {X -0.050,Y -520.337,Z 1308.757,A 0.000,B 0.000,C 90.000,E1 352.299} C_DIS
LIN {X -0.137,Y -523.321,Z 1308.752,A 0.000,B 0.000,C 90.000,E1 351.432} C_DIS
LIN {X -0.132,Y -524.303,Z 1308.751,A 0.000,B 0.000,C 90.000,E1 351.141} C_DIS
LIN {X -0.161,Y -527.703,Z 1308.744,A 0.000,B 0.000,C 90.000,E1 349.982} C_DIS
LIN {X -0.082,Y -530.064,Z 1308.740,A 0.000,B 0.000,C 90.000,E1 349.106} C_DIS
LIN {X -0.013,Y -531.514,Z 1308.736,A 0.000,B 0.000,C 90.000,E1 348.522} C_DIS
LIN {X 0.155,Y -534.003,Z 1308.730,A 0.000,B 0.000,C 90.000,E1 347.353} C_DIS
LIN {X -0.096,Y -535.651,Z 1308.725,A 0.000,B 0.000,C 90.000,E1 346.520} C_DIS
LIN {X 0.122,Y -537.463,Z 1308.719,A 0.000,B 0.000,C 90.000,E1 345.353} C_DIS
LIN {X -0.087,Y -538.591,Z 1308.714,A 0.000,B 0.000,C 90.000,E1 344.519} C_DIS
LIN {X -0.284,Y -539.354,Z 1308.709,A 0.000,B 0.000,C 90.000,E1 343.685} C_DIS
LIN {X -0.257,Y -540.151,Z 1308.703,A 0.000,B 0.000,C 90.000,E1 342.543} C_DIS
LIN {X 0.241,Y -540.381,Z 1308.698,A 0.000,B 0.000,C 90.000,E1 341.638} C_DIS
LIN {X 0.232,Y -540.196,Z 1308.693,A 0.000,B 0.000,C 90.000,E1 340.786} C_DIS
LIN {X 0.223,Y -539.886,Z 1308.689,A 0.000,B 0.000,C 90.000,E1 339.934} C_DIS
LIN {X -0.017,Y -539.482,Z 1308.686,A 0.000,B 0.000,C 90.000,E1 339.390} C_DIS
LIN {X -0.069,Y -538.938,Z 1308.682,A 0.000,B 0.000,C 90.000,E1 338.827} C_DIS
LIN {X 0.123,Y -537.487,Z 1308.676,A 0.000,B 0.000,C 90.000,E1 337.667} C_DIS
LIN {X 0.063,Y -536.576,Z 1308.673,A 0.000,B 0.000,C 90.000,E1 337.102} C_DIS
LIN {X 0.277,Y -535.920,Z 1308.671,A 0.000,B 0.000,C 90.000,E1 336.794} C_DIS
LIN {X -0.002,Y -535.437,Z 1308.670,A 0.000,B 0.000,C 90.000,E1 336.538} C_DIS
LIN {X 0.131,Y -533.350,Z 1308.665,A 0.000,B 0.000,C 90.000,E1 335.665} C_DIS
LIN {X -0.244,Y -530.993,Z 1308.660,A 0.000,B 0.000,C 90.000,E1 334.845} C_DIS
LIN {X -0.062,Y -526.379,Z 1308.652,A 0.000,B 0.000,C 90.000,E1 333.384} C_DIS
LIN {X 0.191,Y -523.595,Z 1308.647,A 0.000,B 0.000,C 90.000,E1 332.487} C_DIS
LIN {X 0.082,Y -519.608,Z 1308.641,A 0.000,B 0.000,C 90.000,E1 331.335} C_DIS
LIN {X 0.046,Y -516.416,Z 1308.636,A 0.000,B 0.000,C 90.000,E1 330.461} C_DIS
LIN {X 0.071,Y -514.174,Z 1308.633,A 0.000,B 0.000,C 90.000,E1 329.871} C_DIS
LIN {X -0.043,Y -507.902,Z 1308.625,A 0.000,B 0.000,C 90.000,E1 328.408} C_DIS
LIN {X -0.130,Y -500.188,Z 1308.615,A 0.000,B 0.000,C 90.000,E1 326.628} C_DIS
LIN {X 0.036,Y -497.921,Z 1308.611,A 0.000,B 0.000,C 90.000,E1 326.008} C_DIS
LIN {X 0.186,Y -496.249,Z 1308.608,A 0.000,B 0.000,C 90.000,E1 325.388} C_DIS
LIN {X 0.179,Y -494.400,Z 1308.603,A 0.000,B 0.000,C 90.000,E1 324.482} C_DIS
LIN {X 0.149,Y -493.162,Z 1308.598,A 0.000,B 0.000,C 90.000,E1 323.577} C_DIS
LIN {X -0.056,Y -491.736,Z 1308.588,A 0.000,B 0.000,C 90.000,E1 321.778} C_DIS
LIN {X -0.210,Y -491.289,Z 1308.583,A 0.000,B 0.000,C 90.000,E1 320.884} C_DIS
LIN {X -0.208,Y -490.847,Z 1308.579,A 0.000,B 0.000,C 90.000,E1 320.275} C_DIS
LIN {X 0.167,Y -490.151,Z 1308.576,A 0.000,B 0.000,C 90.000,E1 319.622} C_DIS
LIN {X 0.161,Y -489.098,Z 1308.573,A 0.000,B 0.000,C 90.000,E1 319.013} C_DIS
LIN {X -0.005,Y -488.310,Z 1308.571,A 0.000,B 0.000,C 90.000,E1 318.728} C_DIS
LIN {X 0.148,Y -487.196,Z 1308.569,A 0.000,B 0.000,C 90.000,E1 318.405} C_DIS
LIN {X 0.224,Y -486.354,Z 1308.568,A 0.000,B 0.000,C 90.000,E1 318.243} C_DIS
LIN {X -0.057,Y -480.779,Z 1308.565,A 0.000,B 0.000,C 90.000,E1 317.676} C_DIS
LIN {X 0.114,Y -459.587,Z 1308.552,A 0.000,B 0.000,C 90.000,E1 315.243} C_DIS
LIN {X -0.078,Y -440.893,Z 1308.538,A 0.000,B 0.000,C 90.000,E1 312.852} C_DIS
LIN {X -0.162,Y -423.927,Z 1308.524,A 0.000,B 0.000,C 90.000,E1 310.378} C_DIS
LIN {X -0.037,Y -408.587,Z 1308.510,A 0.000,B 0.000,C 90.000,E1 307.810} C_DIS
LIN {X 0.043,Y -394.765,Z 1308.496,A 0.000,B 0.000,C 90.000,E1 305.185} C_DIS
LIN {X 0.031,Y -391.351,Z 1308.492,A 0.000,B 0.000,C 90.000,E1 304.485} C_DIS
LIN {X -0.007,Y -391.351,Z 1308.492,A 0.000,B 0.000,C 90.000,E1 304.485} C_DIS
LIN {X -0.061,Y -396.425,Z 1308.461,A 0.000,B 0.000,C 90.000,E1 298.999} C_DIS
LIN {X 0.155,Y -396.883,Z 1308.459,A 0.000,B 0.000,C 90.000,E1 298.615} C_DIS
LIN {X 0.059,Y -397.305,Z 1308.455,A 0.000,B 0.000,C 90.000,E1 297.924} C_DIS
LIN {X 0.166,Y -401.628,Z 1308.426,A 0.000,B 0.000,C 90.000,E1 292.642} C_DIS
LIN {X -0.084,Y -404.698,Z 1308.395,A 0.000,B 0.000,C 90.000,E1 287.094} C_DIS
LIN {X -0.095,Y -404.887,Z 1308.381,A 0.000,B 0.000,C 90.000,E1 284.662} C_DIS
LIN {X -0.092,Y -406.126,Z 1308.364,A 0.000,B 0.000,C 90.000,E1 281.535} C_DIS
LIN {X -0.060,Y -405.827,Z 1308.358,A 0.000,B 0.000,C 90.000,E1 280.489} C_DIS
LIN {X 0.000,Y -405.688,Z 1308.333,A 0.000,B 0.000,C 90.000,E1 275.967} C_DIS
LIN {X 0.038,Y -403.470,Z 1308.304,A 0.000,B 0.000,C 90.000,E1 270.745} C_DIS
LIN {X 0.006,Y -403.257,Z 1308.302,A 0.000,B 0.000,C 90.000,E1 270.401} C_DIS
LIN {X 0.185,Y -398.881,Z 1308.271,A 0.000,B 0.000,C 90.000,E1 264.780} C_DIS
LIN {X 0.082,Y -393.353,Z 1308.244,A 0.000,B 0.000,C 90.000,E1 259.859} C_DIS
LIN {X 0.004,Y -392.783,Z 1308.240,A 0.000,B 0.000,C 90.000,E1 259.162} C_DIS
LIN {X 0.082,Y -386.331,Z 1308.214,A 0.000,B 0.000,C 90.000,E1 254.519} C_DIS
LIN {X 0.044,Y -385.224,Z 1308.208,A 0.000,B 0.000,C 90.000,E1 253.449} C_DIS
LIN {X 0.084,Y -384.028,Z 1308.204,A 0.000,B 0.000,C 90.000,E1 252.725} C_DIS
LIN {X -0.087,Y -377.457,Z 1308.180,A 0.000,B 0.000,C 90.000,E1 248.411} C_DIS
LIN {X 0.005,Y -376.184,Z 1308.174,A 0.000,B 0.000,C 90.000,E1 247.305} C_DIS
LIN {X -0.007,Y -368.355,Z 1308.147,A 0.000,B 0.000,C 90.000,E1 242.538} C_DIS
LIN {X 0.076,Y -367.209,Z 1308.143,A 0.000,B 0.000,C 90.000,E1 241.641} C_DIS
LIN {X 0.039,Y -367.227,Z 1308.143,A 0.000,B 0.000,C 90.000,E1 241.641} C_DIS
LIN {X -0.110,Y -377.939,Z 1308.127,A 0.000,B 0.000,C 90.000,E1 238.869} C_DIS
LIN {X 0.065,Y -389.846,Z 1308.112,A 0.000,B 0.000,C 90.000,E1 236.135} C_DIS
LIN {X -0.029,Y -403.155,Z 1308.097,A 0.000,B 0.000,C 90.000,E1 233.497} C_DIS
LIN {X 0.123,Y -417.959,Z 1308.083,A 0.000,B 0.000,C 90.000,E1 230.884} C_DIS
LIN {X 0.045,Y -434.364,Z 1308.069,A 0.000,B 0.000,C 90.000,E1 228.366} C_DIS
LIN {X 0.174,Y -446.217,Z 1308.060,A 0.000,B 0.000,C 90.000,E1 226.701} C_DIS
LIN {X 0.166,Y -447.045,Z 1308.059,A 0.000,B 0.000,C 90.000,E1 226.539} C_DIS
LIN {X 0.158,Y -447.641,Z 1308.058,A 0.000,B 0.000,C 90.000,E1 226.377} C_DIS
LIN {X 0.150,Y -448.508,Z 1308.056,A 0.000,B 0.000,C 90.000,E1 226.053} C_DIS
LIN {X 0.145,Y -449.139,Z 1308.054,A 0.000,B 0.000,C 90.000,E1 225.729} C_DIS
LIN {X 0.145,Y -450.001,Z 1308.051,A 0.000,B 0.000,C 90.000,E1 225.081} C_DIS
LIN {X 0.152,Y -450.536,Z 1308.047,A 0.000,B 0.000,C 90.000,E1 224.433} C_DIS
LIN {X 0.169,Y -450.931,Z 1308.042,A 0.000,B 0.000,C 90.000,E1 223.461} C_DIS
LIN {X -0.072,Y -451.188,Z 1308.031,A 0.000,B 0.000,C 90.000,E1 221.553} C_DIS
LIN {X -0.182,Y -452.807,Z 1308.011,A 0.000,B 0.000,C 90.000,E1 218.016} C_DIS
LIN {X -0.043,Y -453.803,Z 1308.004,A 0.000,B 0.000,C 90.000,E1 216.710} C_DIS
LIN {X 0.029,Y -455.431,Z 1307.993,A 0.000,B 0.000,C 90.000,E1 214.771} C_DIS
LIN {X -0.012,Y -457.951,Z 1307.979,A 0.000,B 0.000,C 90.000,E1 212.212} C_DIS
LIN {X -0.059,Y -461.740,Z 1307.961,A 0.000,B 0.000,C 90.000,E1 209.027} C_DIS
LIN {X -0.064,Y -465.222,Z 1307.947,A 0.000,B 0.000,C 90.000,E1 206.488} C_DIS
LIN {X 0.031,Y -468.907,Z 1307.933,A 0.000,B 0.000,C 90.000,E1 203.951} C_DIS
LIN {X -0.111,Y -471.946,Z 1307.921,A 0.000,B 0.000,C 90.000,E1 201.770} C_DIS
LIN {X -0.048,Y -474.621,Z 1307.911,A 0.000,B 0.000,C 90.000,E1 199.885} C_DIS
LIN {X 0.085,Y -477.440,Z 1307.900,A 0.000,B 0.000,C 90.000,E1 198.000} C_DIS
LIN {X 0.122,Y -480.170,Z 1307.890,A 0.000,B 0.000,C 90.000,E1 196.134} C_DIS
LIN {X 0.115,Y -482.032,Z 1307.883,A 0.000,B 0.000,C 90.000,E1 194.898} C_DIS
LIN {X -0.002,Y -484.769,Z 1307.873,A 0.000,B 0.000,C 90.000,E1 193.063} C_DIS
LIN {X -0.180,Y -487.396,Z 1307.862,A 0.000,B 0.000,C 90.000,E1 191.243} C_DIS
LIN {X 0.192,Y -489.602,Z 1307.854,A 0.000,B 0.000,C 90.000,E1 189.670} C_DIS
LIN {X -0.067,Y -492.207,Z 1307.844,A 0.000,B 0.000,C 90.000,E1 187.871} C_DIS
LIN {X -0.238,Y -494.336,Z 1307.835,A 0.000,B 0.000,C 90.000,E1 186.372} C_DIS
LIN {X 0.079,Y -496.388,Z 1307.827,A 0.000,B 0.000,C 90.000,E1 184.821} C_DIS
LIN {X -0.053,Y -498.179,Z 1307.818,A 0.000,B 0.000,C 90.000,E1 183.326} C_DIS
LIN {X 0.205,Y -498.872,Z 1307.815,A 0.000,B 0.000,C 90.000,E1 182.694} C_DIS
LIN {X 0.081,Y -500.390,Z 1307.807,A 0.000,B 0.000,C 90.000,E1 181.203} C_DIS
LIN {X -0.024,Y -501.700,Z 1307.798,A 0.000,B 0.000,C 90.000,E1 179.714} C_DIS
LIN {X 0.008,Y -502.500,Z 1307.792,A 0.000,B 0.000,C 90.000,E1 178.511} C_DIS
LIN {X 0.063,Y -503.082,Z 1307.785,A 0.000,B 0.000,C 90.000,E1 177.306} C_DIS
LIN {X 0.127,Y -503.407,Z 1307.778,A 0.000,B 0.000,C 90.000,E1 176.102} C_DIS
LIN {X 0.231,Y -503.465,Z 1307.772,A 0.000,B 0.000,C 90.000,E1 174.894} C_DIS
LIN {X -0.163,Y -503.175,Z 1307.765,A 0.000,B 0.000,C 90.000,E1 173.742} C_DIS
LIN {X 0.067,Y -502.854,Z 1307.760,A 0.000,B 0.000,C 90.000,E1 172.818} C_DIS
LIN {X 0.225,Y -501.915,Z 1307.754,A 0.000,B 0.000,C 90.000,E1 171.602} C_DIS
LIN {X 0.011,Y -501.290,Z 1307.750,A 0.000,B 0.000,C 90.000,E1 171.027} C_DIS
LIN {X -0.199,Y -500.179,Z 1307.745,A 0.000,B 0.000,C 90.000,E1 170.151} C_DIS
LIN {X 0.074,Y -498.694,Z 1307.740,A 0.000,B 0.000,C 90.000,E1 169.218} C_DIS
LIN {X -0.157,Y -496.955,Z 1307.735,A 0.000,B 0.000,C 90.000,E1 168.342} C_DIS
LIN {X 0.076,Y -494.904,Z 1307.730,A 0.000,B 0.000,C 90.000,E1 167.409} C_DIS
LIN {X -0.091,Y -492.651,Z 1307.725,A 0.000,B 0.000,C 90.000,E1 166.520} C_DIS
LIN {X 0.093,Y -489.160,Z 1307.718,A 0.000,B 0.000,C 90.000,E1 165.283} C_DIS
LIN {X -0.258,Y -485.124,Z 1307.712,A 0.000,B 0.000,C 90.000,E1 164.102} C_DIS
LIN {X 0.068,Y -481.354,Z 1307.706,A 0.000,B 0.000,C 90.000,E1 163.142} C_DIS
LIN {X 0.060,Y -479.926,Z 1307.705,A 0.000,B 0.000,C 90.000,E1 162.834} C_DIS
LIN {X -0.279,Y -475.226,Z 1307.700,A 0.000,B 0.000,C 90.000,E1 161.945} C_DIS
LIN {X 0.276,Y -469.714,Z 1307.693,A 0.000,B 0.000,C 90.000,E1 160.786} C_DIS
LIN {X -0.169,Y -467.845,Z 1307.691,A 0.000,B 0.000,C 90.000,E1 160.369} C_DIS
LIN {X 0.166,Y -465.787,Z 1307.687,A 0.000,B 0.000,C 90.000,E1 159.699} C_DIS
LIN {X 0.109,Y -464.908,Z 1307.686,A 0.000,B 0.000,C 90.000,E1 159.390} C_DIS
LIN {X 0.048,Y -464.322,Z 1307.684,A 0.000,B 0.000,C 90.000,E1 159.082} C_DIS
LIN {X -0.081,Y -463.912,Z 1307.680,A 0.000,B 0.000,C 90.000,E1 158.465} C_DIS
LIN {X 0.102,Y -463.929,Z 1307.679,A 0.000,B 0.000,C 90.000,E1 158.284} C_DIS
LIN {X 0.035,Y -464.649,Z 1307.678,A 0.000,B 0.000,C 90.000,E1 157.975} C_DIS
LIN {X 0.217,Y -465.704,Z 1307.677,A 0.000,B 0.000,C 90.000,E1 157.794} C_DIS
LIN {X -0.008,Y -467.313,Z 1307.675,A 0.000,B 0.000,C 90.000,E1 157.486} C_DIS
LIN {X 0.095,Y -470.290,Z 1307.673,A 0.000,B 0.000,C 90.000,E1 157.177} C_DIS
LIN {X -0.060,Y -471.674,Z 1307.672,A 0.000,B 0.000,C 90.000,E1 157.050} C_DIS
LIN {X -0.076,Y -483.930,Z 1307.667,A 0.000,B 0.000,C 90.000,E1 156.049} C_DIS
LIN {X 0.024,Y -489.831,Z 1307.664,A 0.000,B 0.000,C 90.000,E1 155.537} C_DIS
LIN {X 0.038,Y -494.205,Z 1307.662,A 0.000,B 0.000,C 90.000,E1 155.153} C_DIS
LIN {X -0.020,Y -500.826,Z 1307.659,A 0.000,B 0.000,C 90.000,E1 154.537} C_DIS
LIN {X -0.199,Y -504.984,Z 1307.656,A 0.000,B 0.000,C 90.000,E1 154.152} C_DIS
LIN {X -0.042,Y -511.405,Z 1307.652,A 0.000,B 0.000,C 90.000,E1 153.435} C_DIS
LIN {X -0.036,Y -515.202,Z 1307.650,A 0.000,B 0.000,C 90.000,E1 152.999} C_DIS
LIN {X -0.025,Y -519.873,Z 1307.647,A 0.000,B 0.000,C 90.000,E1 152.410} C_DIS
LIN {X 0.024,Y -524.075,Z 1307.644,A 0.000,B 0.000,C 90.000,E1 151.820} C_DIS
LIN {X -0.148,Y -527.687,Z 1307.640,A 0.000,B 0.000,C 90.000,E1 151.257} C_DIS
LIN {X -0.044,Y -530.707,Z 1307.637,A 0.000,B 0.000,C 90.000,E1 150.667} C_DIS
LIN {X 0.083,Y -533.200,Z 1307.634,A 0.000,B 0.000,C 90.000,E1 150.078} C_DIS
LIN {X -0.236,Y -535.251,Z 1307.631,A 0.000,B 0.000,C 90.000,E1 149.537} C_DIS
LIN {X 0.208,Y -536.220,Z 1307.629,A 0.000,B 0.000,C 90.000,E1 149.203} C_DIS
LIN {X -0.090,Y -538.415,Z 1307.624,A 0.000,B 0.000,C 90.000,E1 148.377} C_DIS
LIN {X 0.088,Y -539.724,Z 1307.621,A 0.000,B 0.000,C 90.000,E1 147.788} C_DIS
LIN {X -0.169,Y -541.267,Z 1307.616,A 0.000,B 0.000,C 90.000,E1 146.962} C_DIS
LIN {X 0.068,Y -542.937,Z 1307.610,A 0.000,B 0.000,C 90.000,E1 145.801} C_DIS
LIN {X 0.095,Y -543.699,Z 1307.609,A 0.000,B 0.000,C 90.000,E1 145.515} C_DIS
LIN {X -0.100,Y -544.260,Z 1307.607,A 0.000,B 0.000,C 90.000,E1 145.182} C_DIS
LIN {X 0.268,Y -545.466,Z 1307.605,A 0.000,B 0.000,C 90.000,E1 144.895} C_DIS
LIN {X -0.121,Y -549.122,Z 1307.604,A 0.000,B 0.000,C 90.000,E1 144.689} C_DIS
LIN {X 0.096,Y -550.936,Z 1307.603,A 0.000,B 0.000,C 90.000,E1 144.562} C_DIS
LIN {X -0.012,Y -560.437,Z 1307.601,A 0.000,B 0.000,C 90.000,E1 144.196} C_DIS
LIN {X -0.053,Y -566.521,Z 1307.599,A 0.000,B 0.000,C 90.000,E1 143.909} C_DIS
LIN {X 0.185,Y -572.760,Z 1307.598,A 0.000,B 0.000,C 90.000,E1 143.543} C_DIS
LIN {X 0.004,Y -577.160,Z 1307.596,A 0.000,B 0.000,C 90.000,E1 143.290} C_DIS
LIN {X -0.066,Y -581.475,Z 1307.594,A 0.000,B 0.000,C 90.000,E1 143.004} C_DIS
LIN {X 0.238,Y -587.180,Z 1307.592,A 0.000,B 0.000,C 90.000,E1 142.557} C_DIS
LIN {X 0.151,Y -592.557,Z 1307.590,A 0.000,B 0.000,C 90.000,E1 142.110} C_DIS
LIN {X 0.212,Y -596.502,Z 1307.588,A 0.000,B 0.000,C 90.000,E1 141.743} C_DIS
LIN {X 0.113,Y -600.226,Z 1307.586,A 0.000,B 0.000,C 90.000,E1 141.376} C_DIS
LIN {X -0.171,Y -604.875,Z 1307.583,A 0.000,B 0.000,C 90.000,E1 140.884} C_DIS
LIN {X -0.120,Y -609.178,Z 1307.580,A 0.000,B 0.000,C 90.000,E1 140.356} C_DIS
LIN {X -0.036,Y -613.134,Z 1307.577,A 0.000,B 0.000,C 90.000,E1 139.828} C_DIS
LIN {X -0.091,Y -618.508,Z 1307.573,A 0.000,B 0.000,C 90.000,E1 139.057} C_DIS
LIN {X 0.011,Y -622.613,Z 1307.569,A 0.000,B 0.000,C 90.000,E1 138.405} C_DIS
LIN {X 0.187,Y -625.773,Z 1307.566,A 0.000,B 0.000,C 90.000,E1 137.877} C_DIS
LIN {X 0.178,Y -630.775,Z 1307.561,A 0.000,B 0.000,C 90.000,E1 136.986} C_DIS
LIN {X 0.301,Y -634.935,Z 1307.557,A 0.000,B 0.000,C 90.000,E1 136.215} C_DIS
LIN {X 0.240,Y -642.128,Z 1307.549,A 0.000,B 0.000,C 90.000,E1 134.838} C_DIS
LIN {X 0.368,Y -647.706,Z 1307.543,A 0.000,B 0.000,C 90.000,E1 133.704} C_DIS
LIN {X -0.357,Y -653.775,Z 1307.536,A 0.000,B 0.000,C 90.000,E1 132.528} C_DIS
LIN {X -0.074,Y -659.615,Z 1307.529,A 0.000,B 0.000,C 90.000,E1 131.272} C_DIS
LIN {X -0.122,Y -664.138,Z 1307.524,A 0.000,B 0.000,C 90.000,E1 130.297} C_DIS
LIN {X -0.027,Y -669.326,Z 1307.517,A 0.000,B 0.000,C 90.000,E1 129.072} C_DIS
LIN {X 0.052,Y -673.973,Z 1307.510,A 0.000,B 0.000,C 90.000,E1 127.855} C_DIS
LIN {X 0.172,Y -675.727,Z 1307.508,A 0.000,B 0.000,C 90.000,E1 127.363} C_DIS
LIN {X -0.090,Y -678.970,Z 1307.502,A 0.000,B 0.000,C 90.000,E1 126.423} C_DIS
LIN {X 0.235,Y -681.845,Z 1307.497,A 0.000,B 0.000,C 90.000,E1 125.438} C_DIS
LIN {X 0.211,Y -684.471,Z 1307.492,A 0.000,B 0.000,C 90.000,E1 124.485} C_DIS
LIN {X 0.033,Y -686.257,Z 1307.488,A 0.000,B 0.000,C 90.000,E1 123.785} C_DIS
LIN {X -0.133,Y -687.862,Z 1307.484,A 0.000,B 0.000,C 90.000,E1 123.086} C_DIS
LIN {X -0.075,Y -689.697,Z 1307.479,A 0.000,B 0.000,C 90.000,E1 122.133} C_DIS
LIN {X 0.002,Y -691.319,Z 1307.473,A 0.000,B 0.000,C 90.000,E1 121.180} C_DIS
LIN {X 0.219,Y -693.421,Z 1307.465,A 0.000,B 0.000,C 90.000,E1 119.745} C_DIS
LIN {X 0.242,Y -694.742,Z 1307.459,A 0.000,B 0.000,C 90.000,E1 118.565} C_DIS
LIN {X -0.229,Y -695.284,Z 1307.455,A 0.000,B 0.000,C 90.000,E1 117.897} C_DIS
LIN {X 0.109,Y -695.732,Z 1307.448,A 0.000,B 0.000,C 90.000,E1 116.693} C_DIS
LIN {X -0.115,Y -695.582,Z 1307.443,A 0.000,B 0.000,C 90.000,E1 115.771} C_DIS
LIN {X 0.095,Y -695.277,Z 1307.441,A 0.000,B 0.000,C 90.000,E1 115.283} C_DIS
LIN {X -0.028,Y -694.733,Z 1307.438,A 0.000,B 0.000,C 90.000,E1 114.823} C_DIS
LIN {X 0.185,Y -693.941,Z 1307.435,A 0.000,B 0.000,C 90.000,E1 114.335} C_DIS
LIN {X -0.235,Y -692.445,Z 1307.433,A 0.000,B 0.000,C 90.000,E1 113.898} C_DIS
LIN {X 0.009,Y -691.409,Z 1307.431,A 0.000,B 0.000,C 90.000,E1 113.643} C_DIS
LIN {X 0.208,Y -688.610,Z 1307.429,A 0.000,B 0.000,C 90.000,E1 113.153} C_DIS
LIN {X -0.311,Y -687.581,Z 1307.428,A 0.000,B 0.000,C 90.000,E1 113.078} C_DIS
LIN {X -0.335,Y -681.190,Z 1307.425,A 0.000,B 0.000,C 90.000,E1 112.589} C_DIS
LIN {X -0.053,Y -679.031,Z 1307.425,A 0.000,B 0.000,C 90.000,E1 112.461} C_DIS
LIN {X 0.312,Y -672.642,Z 1307.424,A 0.000,B 0.000,C 90.000,E1 112.206} C_DIS
LIN {X 0.081,Y -664.359,Z 1307.423,A 0.000,B 0.000,C 90.000,E1 112.078} C_DIS
LIN {X -0.103,Y -656.580,Z 1307.422,A 0.000,B 0.000,C 90.000,E1 112.025} C_DIS
LIN {X 0.108,Y -648.946,Z 1307.422,A 0.000,B 0.000,C 90.000,E1 111.972} C_DIS
LIN {X 0.219,Y -643.874,Z 1307.422,A 0.000,B 0.000,C 90.000,E1 111.897} C_DIS
LIN {X 0.031,Y -641.813,Z 1307.421,A 0.000,B 0.000,C 90.000,E1 111.844} C_DIS
LIN {X -0.011,Y -641.772,Z 1307.421,A 0.000,B 0.000,C 90.000,E1 111.844} C_DIS
LIN {X -0.092,Y -643.341,Z 1307.420,A 0.000,B 0.000,C 90.000,E1 111.535} C_DIS
LIN {X -0.112,Y -651.133,Z 1307.414,A 0.000,B 0.000,C 90.000,E1 110.536} C_DIS
LIN {X -0.358,Y -655.384,Z 1307.411,A 0.000,B 0.000,C 90.000,E1 109.939} C_DIS
LIN {X 0.328,Y -659.681,Z 1307.406,A 0.000,B 0.000,C 90.000,E1 109.141} C_DIS
LIN {X 0.107,Y -662.233,Z 1307.404,A 0.000,B 0.000,C 90.000,E1 108.671} C_DIS
LIN {X 0.020,Y -665.515,Z 1307.400,A 0.000,B 0.000,C 90.000,E1 107.946} C_DIS
LIN {X -0.040,Y -668.424,Z 1307.396,A 0.000,B 0.000,C 90.000,E1 107.221} C_DIS
LIN {X -0.001,Y -670.104,Z 1307.393,A 0.000,B 0.000,C 90.000,E1 106.732} C_DIS
LIN {X -0.213,Y -672.285,Z 1307.389,A 0.000,B 0.000,C 90.000,E1 106.024} C_DIS
LIN {X -0.220,Y -674.081,Z 1307.385,A 0.000,B 0.000,C 90.000,E1 105.300} C_DIS
LIN {X 0.263,Y -675.589,Z 1307.381,A 0.000,B 0.000,C 90.000,E1 104.537} C_DIS
LIN {X 0.111,Y -676.868,Z 1307.377,A 0.000,B 0.000,C 90.000,E1 103.828} C_DIS
LIN {X -0.030,Y -677.726,Z 1307.373,A 0.000,B 0.000,C 90.000,E1 103.119} C_DIS
LIN {X -0.165,Y -678.192,Z 1307.369,A 0.000,B 0.000,C 90.000,E1 102.411} C_DIS
LIN {X 0.267,Y -678.334,Z 1307.366,A 0.000,B 0.000,C 90.000,E1 101.895} C_DIS
LIN {X 0.181,Y -678.290,Z 1307.364,A 0.000,B 0.000,C 90.000,E1 101.422} C_DIS
LIN {X 0.089,Y -678.041,Z 1307.361,A 0.000,B 0.000,C 90.000,E1 100.950} C_DIS
LIN {X -0.179,Y -677.314,Z 1307.357,A 0.000,B 0.000,C 90.000,E1 100.254} C_DIS
LIN {X 0.383,Y -676.584,Z 1307.354,A 0.000,B 0.000,C 90.000,E1 99.726} C_DIS
LIN {X 0.158,Y -675.525,Z 1307.352,A 0.000,B 0.000,C 90.000,E1 99.265} C_DIS
LIN {X -0.068,Y -674.151,Z 1307.349,A 0.000,B 0.000,C 90.000,E1 98.803} C_DIS
LIN {X -0.300,Y -672.343,Z 1307.346,A 0.000,B 0.000,C 90.000,E1 98.341} C_DIS
LIN {X 0.217,Y -670.315,Z 1307.344,A 0.000,B 0.000,C 90.000,E1 97.814} C_DIS
LIN {X 0.049,Y -668.613,Z 1307.342,A 0.000,B 0.000,C 90.000,E1 97.466} C_DIS
LIN {X 0.153,Y -663.440,Z 1307.336,A 0.000,B 0.000,C 90.000,E1 96.486} C_DIS
LIN {X -0.148,Y -660.617,Z 1307.333,A 0.000,B 0.000,C 90.000,E1 96.024} C_DIS
LIN {X 0.088,Y -656.553,Z 1307.330,A 0.000,B 0.000,C 90.000,E1 95.391} C_DIS
LIN {X -0.314,Y -653.101,Z 1307.327,A 0.000,B 0.000,C 90.000,E1 94.935} C_DIS
LIN {X -0.137,Y -648.215,Z 1307.324,A 0.000,B 0.000,C 90.000,E1 94.302} C_DIS
LIN {X 0.110,Y -644.031,Z 1307.321,A 0.000,B 0.000,C 90.000,E1 93.784} C_DIS
LIN {X 0.188,Y -636.227,Z 1307.316,A 0.000,B 0.000,C 90.000,E1 92.922} C_DIS
LIN {X 0.092,Y -629.038,Z 1307.312,A 0.000,B 0.000,C 90.000,E1 92.178} C_DIS
LIN {X -0.286,Y -624.052,Z 1307.309,A 0.000,B 0.000,C 90.000,E1 91.718} C_DIS
LIN {X 0.286,Y -616.071,Z 1307.306,A 0.000,B 0.000,C 90.000,E1 90.974} C_DIS
LIN {X -0.004,Y -608.388,Z 1307.303,A 0.000,B 0.000,C 90.000,E1 90.458} C_DIS
LIN {X 0.120,Y -602.031,Z 1307.300,A 0.000,B 0.000,C 90.000,E1 90.057} C_DIS
LIN {X -0.257,Y -597.005,Z 1307.299,A 0.000,B 0.000,C 90.000,E1 89.828} C_DIS
LIN {X 0.282,Y -592.063,Z 1307.298,A 0.000,B 0.000,C 90.000,E1 89.542} C_DIS
LIN {X -0.135,Y -588.512,Z 1307.297,A 0.000,B 0.000,C 90.000,E1 89.427} C_DIS
LIN {X -0.105,Y -576.283,Z 1307.294,A 0.000,B 0.000,C 90.000,E1 88.969} C_DIS
LIN {X -0.261,Y -572.189,Z 1307.293,A 0.000,B 0.000,C 90.000,E1 88.797} C_DIS
LIN {X 0.264,Y -572.116,Z 1307.293,A 0.000,B 0.000,C 90.000,E1 88.740} C_DIS
LIN {X 0.160,Y -570.502,Z 1307.292,A 0.000,B 0.000,C 90.000,E1 88.511} C_DIS
LIN {X 0.118,Y -570.485,Z 1307.292,A 0.000,B 0.000,C 90.000,E1 88.511} C_DIS
LIN {X -0.175,Y -570.216,Z 1307.290,A 0.000,B 0.000,C 90.000,E1 88.224} C_DIS
LIN {X 0.141,Y -571.099,Z 1307.283,A 0.000,B 0.000,C 90.000,E1 86.963} C_DIS
LIN {X 0.027,Y -573.004,Z 1307.273,A 0.000,B 0.000,C 90.000,E1 85.065} C_DIS
LIN {X -0.162,Y -574.851,Z 1307.264,A 0.000,B 0.000,C 90.000,E1 83.451} C_DIS
LIN {X 0.097,Y -577.403,Z 1307.251,A 0.000,B 0.000,C 90.000,E1 81.254} C_DIS
LIN {X 0.062,Y -579.312,Z 1307.243,A 0.000,B 0.000,C 90.000,E1 79.634} C_DIS
LIN {X 0.043,Y -580.763,Z 1307.235,A 0.000,B 0.000,C 90.000,E1 78.285} C_DIS
LIN {X -0.176,Y -581.785,Z 1307.229,A 0.000,B 0.000,C 90.000,E1 77.229} C_DIS
LIN {X 0.182,Y -582.707,Z 1307.223,A 0.000,B 0.000,C 90.000,E1 76.117} C_DIS
LIN {X -0.205,Y -583.701,Z 1307.216,A 0.000,B 0.000,C 90.000,E1 74.810} C_DIS
LIN {X -0.179,Y -584.755,Z 1307.207,A 0.000,B 0.000,C 90.000,E1 73.196} C_DIS
LIN {X -0.136,Y -585.787,Z 1307.198,A 0.000,B 0.000,C 90.000,E1 71.583} C_DIS
LIN {X 0.300,Y -586.813,Z 1307.189,A 0.000,B 0.000,C 90.000,E1 69.934} C_DIS
LIN {X 0.001,Y -587.876,Z 1307.180,A 0.000,B 0.000,C 90.000,E1 68.358} C_DIS
LIN {X 0.147,Y -588.938,Z 1307.171,A 0.000,B 0.000,C 90.000,E1 66.741} C_DIS
LIN {X -0.082,Y -590.187,Z 1307.161,A 0.000,B 0.000,C 90.000,E1 64.897} C_DIS
LIN {X -0.167,Y -591.319,Z 1307.152,A 0.000,B 0.000,C 90.000,E1 63.307} C_DIS
LIN {X -0.160,Y -593.131,Z 1307.140,A 0.000,B 0.000,C 90.000,E1 61.179} C_DIS
LIN {X -0.357,Y -594.442,Z 1307.132,A 0.000,B 0.000,C 90.000,E1 59.871} C_DIS
LIN {X -0.118,Y -596.353,Z 1307.122,A 0.000,B 0.000,C 90.000,E1 57.995} C_DIS
LIN {X -0.011,Y -598.314,Z 1307.112,A 0.000,B 0.000,C 90.000,E1 56.135} C_DIS
LIN {X -0.236,Y -599.428,Z 1307.106,A 0.000,B 0.000,C 90.000,E1 55.102} C_DIS
LIN {X -0.212,Y -600.665,Z 1307.099,A 0.000,B 0.000,C 90.000,E1 53.783} C_DIS
LIN {X -0.047,Y -602.031,Z 1307.090,A 0.000,B 0.000,C 90.000,E1 52.190} C_DIS
LIN {X -0.358,Y -602.825,Z 1307.084,A 0.000,B 0.000,C 90.000,E1 51.170} C_DIS
LIN {X -0.025,Y -603.762,Z 1307.077,A 0.000,B 0.000,C 90.000,E1 49.828} C_DIS
LIN {X 0.274,Y -604.332,Z 1307.073,A 0.000,B 0.000,C 90.000,E1 49.013} C_DIS
LIN {X -0.080,Y -604.662,Z 1307.067,A 0.000,B 0.000,C 90.000,E1 48.000} C_DIS
LIN {X 0.039,Y -604.911,Z 1307.058,A 0.000,B 0.000,C 90.000,E1 46.419} C_DIS
LIN {X -0.069,Y -604.981,Z 1307.051,A 0.000,B 0.000,C 90.000,E1 45.121} C_DIS
LIN {X -0.001,Y -604.827,Z 1307.045,A 0.000,B 0.000,C 90.000,E1 44.069} C_DIS
LIN {X -0.307,Y -604.445,Z 1307.036,A 0.000,B 0.000,C 90.000,E1 42.528} C_DIS
LIN {X -0.012,Y -604.023,Z 1307.029,A 0.000,B 0.000,C 90.000,E1 41.191} C_DIS
LIN {X -0.058,Y -603.404,Z 1307.022,A 0.000,B 0.000,C 90.000,E1 39.886} C_DIS
LIN {X 0.028,Y -602.898,Z 1307.016,A 0.000,B 0.000,C 90.000,E1 38.830} C_DIS
LIN {X 0.064,Y -602.608,Z 1307.013,A 0.000,B 0.000,C 90.000,E1 38.302} C_DIS
LIN {X 0.002,Y -601.421,Z 1307.006,A 0.000,B 0.000,C 90.000,E1 36.996} C_DIS
LIN {X 0.152,Y -600.164,Z 1307.000,A 0.000,B 0.000,C 90.000,E1 35.931} C_DIS
LIN {X -0.060,Y -598.699,Z 1306.994,A 0.000,B 0.000,C 90.000,E1 34.898} C_DIS
LIN {X -0.053,Y -596.410,Z 1306.987,A 0.000,B 0.000,C 90.000,E1 33.579} C_DIS
LIN {X 0.293,Y -594.661,Z 1306.982,A 0.000,B 0.000,C 90.000,E1 32.752} C_DIS
LIN {X 0.005,Y -592.009,Z 1306.976,A 0.000,B 0.000,C 90.000,E1 31.720} C_DIS
LIN {X -0.015,Y -589.637,Z 1306.972,A 0.000,B 0.000,C 90.000,E1 30.924} C_DIS
LIN {X -0.055,Y -586.987,Z 1306.967,A 0.000,B 0.000,C 90.000,E1 30.129} C_DIS
LIN {X 0.000,Y -585.003,Z 1306.964,A 0.000,B 0.000,C 90.000,E1 29.589} C_DIS
LIN {X -0.247,Y -582.795,Z 1306.961,A 0.000,B 0.000,C 90.000,E1 29.077} C_DIS
LIN {X 0.217,Y -579.730,Z 1306.958,A 0.000,B 0.000,C 90.000,E1 28.359} C_DIS
LIN {X 0.009,Y -577.748,Z 1306.955,A 0.000,B 0.000,C 90.000,E1 27.975} C_DIS
LIN {X 0.262,Y -572.788,Z 1306.950,A 0.000,B 0.000,C 90.000,E1 27.001} C_DIS
LIN {X -0.143,Y -568.845,Z 1306.946,A 0.000,B 0.000,C 90.000,E1 26.360} C_DIS
LIN {X -0.160,Y -563.614,Z 1306.942,A 0.000,B 0.000,C 90.000,E1 25.540} C_DIS
LIN {X 0.104,Y -558.931,Z 1306.938,A 0.000,B 0.000,C 90.000,E1 24.823} C_DIS
LIN {X 0.086,Y -553.716,Z 1306.934,A 0.000,B 0.000,C 90.000,E1 24.131} C_DIS
LIN {X -0.199,Y -548.106,Z 1306.930,A 0.000,B 0.000,C 90.000,E1 23.462} C_DIS
LIN {X -0.305,Y -542.191,Z 1306.926,A 0.000,B 0.000,C 90.000,E1 22.770} C_DIS
LIN {X -0.090,Y -534.690,Z 1306.922,A 0.000,B 0.000,C 90.000,E1 21.897} C_DIS
LIN {X 0.018,Y -530.765,Z 1306.919,A 0.000,B 0.000,C 90.000,E1 21.461} C_DIS
LIN {X 0.023,Y -521.582,Z 1306.914,A 0.000,B 0.000,C 90.000,E1 20.482} C_DIS
LIN {X 0.056,Y -512.321,Z 1306.908,A 0.000,B 0.000,C 90.000,E1 19.504} C_DIS
LIN {X -0.043,Y -501.344,Z 1306.902,A 0.000,B 0.000,C 90.000,E1 18.417} C_DIS
LIN {X 0.054,Y -490.503,Z 1306.896,A 0.000,B 0.000,C 90.000,E1 17.347} C_DIS
LIN {X -0.060,Y -483.302,Z 1306.893,A 0.000,B 0.000,C 90.000,E1 16.677} C_DIS
LIN {X 0.174,Y -473.148,Z 1306.887,A 0.000,B 0.000,C 90.000,E1 15.717} C_DIS
LIN {X -0.125,Y -454.010,Z 1306.878,A 0.000,B 0.000,C 90.000,E1 14.008} C_DIS
LIN {X -0.247,Y -437.974,Z 1306.869,A 0.000,B 0.000,C 90.000,E1 12.479} C_DIS
LIN {X -0.204,Y -422.271,Z 1306.860,A 0.000,B 0.000,C 90.000,E1 10.838} C_DIS
LIN {X -0.095,Y -407.939,Z 1306.851,A 0.000,B 0.000,C 90.000,E1 9.265} C_DIS
LIN {X -0.046,Y -398.322,Z 1306.845,A 0.000,B 0.000,C 90.000,E1 8.163} C_DIS
LIN {X -0.012,Y -397.120,Z 1306.844,A 0.000,B 0.000,C 90.000,E1 7.992} C_DIS
LIN {X -0.046,Y -395.326,Z 1306.843,A 0.000,B 0.000,C 90.000,E1 7.701} C_DIS
LIN {X -0.084,Y -395.323,Z 1306.843,A 0.000,B 0.000,C 90.000,E1 7.701} C_DIS
LIN {X -0.060,Y -395.926,Z 1306.842,A 0.000,B 0.000,C 90.000,E1 7.587} C_DIS
LIN {X 0.158,Y -398.709,Z 1306.841,A 0.000,B 0.000,C 90.000,E1 7.296} C_DIS
LIN {X 0.059,Y -400.289,Z 1306.840,A 0.000,B 0.000,C 90.000,E1 7.182} C_DIS
LIN {X 0.204,Y -411.058,Z 1306.836,A 0.000,B 0.000,C 90.000,E1 6.486} C_DIS
LIN {X -0.072,Y -416.104,Z 1306.834,A 0.000,B 0.000,C 90.000,E1 6.201} C_DIS
LIN {X 0.080,Y -423.966,Z 1306.831,A 0.000,B 0.000,C 90.000,E1 5.625} C_DIS
LIN {X -0.154,Y -431.784,Z 1306.828,A 0.000,B 0.000,C 90.000,E1 5.049} C_DIS
LIN {X 0.061,Y -436.466,Z 1306.826,A 0.000,B 0.000,C 90.000,E1 4.645} C_DIS
LIN {X 0.023,Y -442.536,Z 1306.823,A 0.000,B 0.000,C 90.000,E1 4.131} C_DIS
LIN {X -0.006,Y -451.303,Z 1306.818,A 0.000,B 0.000,C 90.000,E1 3.326} C_DIS
LIN {X -0.039,Y -455.550,Z 1306.816,A 0.000,B 0.000,C 90.000,E1 2.922} C_DIS
LIN {X -0.021,Y -461.283,Z 1306.813,A 0.000,B 0.000,C 90.000,E1 2.350} C_DIS
LIN {X -0.170,Y -466.794,Z 1306.810,A 0.000,B 0.000,C 90.000,E1 1.776} C_DIS
LIN {X 0.003,Y -472.017,Z 1306.806,A 0.000,B 0.000,C 90.000,E1 1.146} C_DIS
LIN {X -0.193,Y -475.406,Z 1306.804,A 0.000,B 0.000,C 90.000,E1 0.745} C_DIS
LIN {X 0.204,Y -479.039,Z 1306.802,A 0.000,B 0.000,C 90.000,E1 0.229} C_DIS
LIN {X 0.145,Y -485.592,Z 1306.796,A 0.000,B 0.000,C 90.000,E1 359.312} C_DIS
LIN {X -0.044,Y -490.611,Z 1306.792,A 0.000,B 0.000,C 90.000,E1 358.568} C_DIS
LIN {X -0.171,Y -495.200,Z 1306.788,A 0.000,B 0.000,C 90.000,E1 357.822} C_DIS
LIN {X 0.040,Y -498.723,Z 1306.784,A 0.000,B 0.000,C 90.000,E1 357.192} C_DIS
LIN {X -0.010,Y -502.765,Z 1306.780,A 0.000,B 0.000,C 90.000,E1 356.445} C_DIS
LIN {X -0.018,Y -506.531,Z 1306.776,A 0.000,B 0.000,C 90.000,E1 355.698} C_DIS
LIN {X 0.008,Y -510.096,Z 1306.772,A 0.000,B 0.000,C 90.000,E1 354.951} C_DIS
LIN {X 0.028,Y -514.703,Z 1306.766,A 0.000,B 0.000,C 90.000,E1 353.913} C_DIS
LIN {X 0.124,Y -517.775,Z 1306.762,A 0.000,B 0.000,C 90.000,E1 353.166} C_DIS
LIN {X 0.012,Y -521.030,Z 1306.757,A 0.000,B 0.000,C 90.000,E1 352.299} C_DIS
LIN {X -0.067,Y -524.047,Z 1306.752,A 0.000,B 0.000,C 90.000,E1 351.432} C_DIS
LIN {X -0.060,Y -525.030,Z 1306.751,A 0.000,B 0.000,C 90.000,E1 351.141} C_DIS
LIN {X -0.078,Y -528.462,Z 1306.744,A 0.000,B 0.000,C 90.000,E1 349.982} C_DIS
LIN {X 0.046,Y -531.543,Z 1306.738,A 0.000,B 0.000,C 90.000,E1 348.814} C_DIS
LIN {X 0.127,Y -532.914,Z 1306.735,A 0.000,B 0.000,C 90.000,E1 348.229} C_DIS
LIN {X -0.207,Y -535.350,Z 1306.728,A 0.000,B 0.000,C 90.000,E1 347.117} C_DIS
LIN {X 0.079,Y -536.935,Z 1306.724,A 0.000,B 0.000,C 90.000,E1 346.228} C_DIS
LIN {X -0.071,Y -538.682,Z 1306.717,A 0.000,B 0.000,C 90.000,E1 345.102} C_DIS
LIN {X 0.259,Y -539.695,Z 1306.713,A 0.000,B 0.000,C 90.000,E1 344.212} C_DIS
LIN {X 0.078,Y -540.447,Z 1306.708,A 0.000,B 0.000,C 90.000,E1 343.378} C_DIS
LIN {X -0.096,Y -540.985,Z 1306.703,A 0.000,B 0.000,C 90.000,E1 342.543} C_DIS
LIN {X -0.103,Y -541.245,Z 1306.698,A 0.000,B 0.000,C 90.000,E1 341.692} C_DIS
LIN {X 0.182,Y -541.250,Z 1306.695,A 0.000,B 0.000,C 90.000,E1 341.094} C_DIS
LIN {X -0.281,Y -540.802,Z 1306.689,A 0.000,B 0.000,C 90.000,E1 340.007} C_DIS
LIN {X -0.097,Y -540.186,Z 1306.684,A 0.000,B 0.000,C 90.000,E1 339.135} C_DIS
LIN {X 0.165,Y -539.527,Z 1306.681,A 0.000,B 0.000,C 90.000,E1 338.539} C_DIS
LIN {X 0.064,Y -538.041,Z 1306.675,A 0.000,B 0.000,C 90.000,E1 337.411} C_DIS
LIN {X 0.010,Y -537.047,Z 1306.671,A 0.000,B 0.000,C 90.000,E1 336.847} C_DIS
LIN {X -0.117,Y -534.483,Z 1306.665,A 0.000,B 0.000,C 90.000,E1 335.717} C_DIS
LIN {X 0.005,Y -532.128,Z 1306.660,A 0.000,B 0.000,C 90.000,E1 334.845} C_DIS
LIN {X 0.092,Y -529.409,Z 1306.656,A 0.000,B 0.000,C 90.000,E1 333.973} C_DIS
LIN {X 0.005,Y -524.733,Z 1306.647,A 0.000,B 0.000,C 90.000,E1 332.538} C_DIS
LIN {X -0.082,Y -520.659,Z 1306.641,A 0.000,B 0.000,C 90.000,E1 331.385} C_DIS
LIN {X -0.101,Y -517.422,Z 1306.636,A 0.000,B 0.000,C 90.000,E1 330.511} C_DIS
LIN {X 0.209,Y -514.538,Z 1306.632,A 0.000,B 0.000,C 90.000,E1 329.744} C_DIS
LIN {X 0.095,Y -508.141,Z 1306.624,A 0.000,B 0.000,C 90.000,E1 328.280} C_DIS
LIN {X 0.204,Y -500.875,Z 1306.615,A 0.000,B 0.000,C 90.000,E1 326.628} C_DIS
LIN {X -0.319,Y -498.603,Z 1306.611,A 0.000,B 0.000,C 90.000,E1 326.087} C_DIS
LIN {X -0.033,Y -497.642,Z 1306.610,A 0.000,B 0.000,C 90.000,E1 325.754} C_DIS
LIN {X -0.026,Y -495.515,Z 1306.605,A 0.000,B 0.000,C 90.000,E1 324.848} C_DIS
LIN {X 0.246,Y -494.038,Z 1306.600,A 0.000,B 0.000,C 90.000,E1 323.909} C_DIS
LIN {X -0.085,Y -492.602,Z 1306.591,A 0.000,B 0.000,C 90.000,E1 322.431} C_DIS
LIN {X 0.310,Y -492.001,Z 1306.584,A 0.000,B 0.000,C 90.000,E1 321.170} C_DIS
LIN {X 0.163,Y -491.837,Z 1306.579,A 0.000,B 0.000,C 90.000,E1 320.275} C_DIS
LIN {X 0.014,Y -491.365,Z 1306.574,A 0.000,B 0.000,C 90.000,E1 319.380} C_DIS
LIN {X 0.019,Y -490.776,Z 1306.571,A 0.000,B 0.000,C 90.000,E1 318.771} C_DIS
LIN {X 0.020,Y -489.855,Z 1306.568,A 0.000,B 0.000,C 90.000,E1 318.162} C_DIS
LIN {X -0.147,Y -489.160,Z 1306.566,A 0.000,B 0.000,C 90.000,E1 317.877} C_DIS
LIN {X 0.012,Y -488.187,Z 1306.564,A 0.000,B 0.000,C 90.000,E1 317.553} C_DIS
LIN {X 0.092,Y -487.502,Z 1306.563,A 0.000,B 0.000,C 90.000,E1 317.391} C_DIS
LIN {X 0.170,Y -486.514,Z 1306.563,A 0.000,B 0.000,C 90.000,E1 317.229} C_DIS
LIN {X -0.071,Y -465.324,Z 1306.549,A 0.000,B 0.000,C 90.000,E1 314.838} C_DIS
LIN {X -0.109,Y -446.818,Z 1306.536,A 0.000,B 0.000,C 90.000,E1 312.447} C_DIS
LIN {X 0.026,Y -430.019,Z 1306.522,A 0.000,B 0.000,C 90.000,E1 309.967} C_DIS
LIN {X 0.007,Y -414.812,Z 1306.508,A 0.000,B 0.000,C 90.000,E1 307.443} C_DIS
LIN {X -0.056,Y -401.099,Z 1306.494,A 0.000,B 0.000,C 90.000,E1 304.865} C_DIS
LIN {X 0.036,Y -392.337,Z 1306.483,A 0.000,B 0.000,C 90.000,E1 303.007} C_DIS
LIN {X -0.001,Y -392.340,Z 1306.483,A 0.000,B 0.000,C 90.000,E1 303.007} C_DIS
LIN {X 0.090,Y -397.036,Z 1306.458,A 0.000,B 0.000,C 90.000,E1 298.487} C_DIS
LIN {X -0.130,Y -401.412,Z 1306.427,A 0.000,B 0.000,C 90.000,E1 292.898} C_DIS
LIN {X 0.107,Y -401.669,Z 1306.425,A 0.000,B 0.000,C 90.000,E1 292.514} C_DIS
LIN {X 0.238,Y -404.763,Z 1306.394,A 0.000,B 0.000,C 90.000,E1 286.913} C_DIS
LIN {X 0.144,Y -406.157,Z 1306.363,A 0.000,B 0.000,C 90.000,E1 281.366} C_DIS
LIN {X -0.156,Y -405.640,Z 1306.334,A 0.000,B 0.000,C 90.000,E1 276.201} C_DIS
LIN {X -0.150,Y -405.648,Z 1306.332,A 0.000,B 0.000,C 90.000,E1 275.853} C_DIS
LIN {X -0.078,Y -403.558,Z 1306.305,A 0.000,B 0.000,C 90.000,E1 270.974} C_DIS
LIN {X -0.143,Y -403.112,Z 1306.302,A 0.000,B 0.000,C 90.000,E1 270.286} C_DIS
LIN {X 0.086,Y -399.039,Z 1306.272,A 0.000,B 0.000,C 90.000,E1 265.008} C_DIS
LIN {X 0.027,Y -398.687,Z 1306.270,A 0.000,B 0.000,C 90.000,E1 264.666} C_DIS
LIN {X -0.090,Y -393.242,Z 1306.243,A 0.000,B 0.000,C 90.000,E1 259.746} C_DIS
LIN {X -0.130,Y -392.971,Z 1306.241,A 0.000,B 0.000,C 90.000,E1 259.398} C_DIS
LIN {X -0.171,Y -392.565,Z 1306.239,A 0.000,B 0.000,C 90.000,E1 259.050} C_DIS
LIN {X -0.011,Y -386.178,Z 1306.213,A 0.000,B 0.000,C 90.000,E1 254.393} C_DIS
LIN {X -0.049,Y -385.072,Z 1306.207,A 0.000,B 0.000,C 90.000,E1 253.323} C_DIS
LIN {X 0.192,Y -378.201,Z 1306.183,A 0.000,B 0.000,C 90.000,E1 248.954} C_DIS
LIN {X -0.088,Y -375.981,Z 1306.173,A 0.000,B 0.000,C 90.000,E1 247.177} C_DIS
LIN {X -0.064,Y -369.271,Z 1306.151,A 0.000,B 0.000,C 90.000,E1 243.204} C_DIS
LIN {X 0.065,Y -369.266,Z 1306.151,A 0.000,B 0.000,C 90.000,E1 243.179} C_DIS
LIN {X -0.046,Y -380.131,Z 1306.135,A 0.000,B 0.000,C 90.000,E1 240.205} C_DIS
LIN {X -0.037,Y -392.247,Z 1306.119,A 0.000,B 0.000,C 90.000,E1 237.327} C_DIS
LIN {X -0.067,Y -405.002,Z 1306.104,A 0.000,B 0.000,C 90.000,E1 234.689} C_DIS
LIN {X -0.115,Y -419.197,Z 1306.089,A 0.000,B 0.000,C 90.000,E1 232.110} C_DIS
LIN {X 0.216,Y -434.928,Z 1306.075,A 0.000,B 0.000,C 90.000,E1 229.542} C_DIS
LIN {X 0.026,Y -446.321,Z 1306.066,A 0.000,B 0.000,C 90.000,E1 227.919} C_DIS
LIN {X 0.016,Y -447.365,Z 1306.065,A 0.000,B 0.000,C 90.000,E1 227.757} C_DIS
LIN {X 0.011,Y -448.056,Z 1306.064,A 0.000,B 0.000,C 90.000,E1 227.595} C_DIS
LIN {X 0.004,Y -448.581,Z 1306.064,A 0.000,B 0.000,C 90.000,E1 227.433} C_DIS
LIN {X 0.024,Y -449.367,Z 1306.062,A 0.000,B 0.000,C 90.000,E1 227.106} C_DIS
LIN {X 0.020,Y -449.950,Z 1306.060,A 0.000,B 0.000,C 90.000,E1 226.782} C_DIS
LIN {X 0.023,Y -450.728,Z 1306.056,A 0.000,B 0.000,C 90.000,E1 226.134} C_DIS
LIN {X 0.035,Y -451.201,Z 1306.053,A 0.000,B 0.000,C 90.000,E1 225.486} C_DIS
LIN {X 0.062,Y -451.520,Z 1306.047,A 0.000,B 0.000,C 90.000,E1 224.514} C_DIS
LIN {X -0.185,Y -451.629,Z 1306.035,A 0.000,B 0.000,C 90.000,E1 222.285} C_DIS
LIN {X -0.219,Y -453.346,Z 1306.012,A 0.000,B 0.000,C 90.000,E1 218.096} C_DIS
LIN {X 0.209,Y -454.080,Z 1306.006,A 0.000,B 0.000,C 90.000,E1 217.076} C_DIS
LIN {X 0.277,Y -455.901,Z 1305.994,A 0.000,B 0.000,C 90.000,E1 214.818} C_DIS
LIN {X 0.112,Y -458.709,Z 1305.978,A 0.000,B 0.000,C 90.000,E1 211.957} C_DIS
LIN {X 0.198,Y -462.162,Z 1305.962,A 0.000,B 0.000,C 90.000,E1 209.077} C_DIS
LIN {X 0.127,Y -466.021,Z 1305.946,A 0.000,B 0.000,C 90.000,E1 206.232} C_DIS
LIN {X 0.107,Y -469.260,Z 1305.934,A 0.000,B 0.000,C 90.000,E1 204.027} C_DIS
LIN {X 0.064,Y -471.465,Z 1305.925,A 0.000,B 0.000,C 90.000,E1 202.461} C_DIS
LIN {X -0.155,Y -474.098,Z 1305.914,A 0.000,B 0.000,C 90.000,E1 200.610} C_DIS
LIN {X -0.062,Y -477.431,Z 1305.902,A 0.000,B 0.000,C 90.000,E1 198.417} C_DIS
LIN {X -0.027,Y -480.213,Z 1305.892,A 0.000,B 0.000,C 90.000,E1 196.551} C_DIS
LIN {X -0.054,Y -482.547,Z 1305.883,A 0.000,B 0.000,C 90.000,E1 195.009} C_DIS
LIN {X -0.169,Y -485.350,Z 1305.873,A 0.000,B 0.000,C 90.000,E1 193.175} C_DIS
LIN {X 0.259,Y -487.577,Z 1305.865,A 0.000,B 0.000,C 90.000,E1 191.591} C_DIS
LIN {X 0.152,Y -489.840,Z 1305.856,A 0.000,B 0.000,C 90.000,E1 190.074} C_DIS
LIN {X 0.004,Y -492.060,Z 1305.848,A 0.000,B 0.000,C 90.000,E1 188.568} C_DIS
LIN {X -0.166,Y -494.250,Z 1305.839,A 0.000,B 0.000,C 90.000,E1 187.068} C_DIS
LIN {X 0.103,Y -496.794,Z 1305.829,A 0.000,B 0.000,C 90.000,E1 185.220} C_DIS
LIN {X 0.109,Y -498.386,Z 1305.822,A 0.000,B 0.000,C 90.000,E1 184.012} C_DIS
LIN {X -0.025,Y -500.142,Z 1305.814,A 0.000,B 0.000,C 90.000,E1 182.522} C_DIS
LIN {X 0.119,Y -501.126,Z 1305.809,A 0.000,B 0.000,C 90.000,E1 181.604} C_DIS
LIN {X 0.027,Y -502.567,Z 1305.801,A 0.000,B 0.000,C 90.000,E1 180.115} C_DIS
LIN {X 0.073,Y -503.522,Z 1305.794,A 0.000,B 0.000,C 90.000,E1 178.912} C_DIS
LIN {X 0.146,Y -504.289,Z 1305.787,A 0.000,B 0.000,C 90.000,E1 177.707} C_DIS
LIN {X 0.120,Y -504.860,Z 1305.779,A 0.000,B 0.000,C 90.000,E1 176.216} C_DIS
LIN {X -0.183,Y -505.003,Z 1305.774,A 0.000,B 0.000,C 90.000,E1 175.355} C_DIS
LIN {X -0.055,Y -504.974,Z 1305.767,A 0.000,B 0.000,C 90.000,E1 174.147} C_DIS
LIN {X 0.003,Y -504.545,Z 1305.759,A 0.000,B 0.000,C 90.000,E1 172.648} C_DIS
LIN {X 0.182,Y -503.661,Z 1305.753,A 0.000,B 0.000,C 90.000,E1 171.432} C_DIS
LIN {X -0.152,Y -502.312,Z 1305.746,A 0.000,B 0.000,C 90.000,E1 170.274} C_DIS
LIN {X 0.142,Y -501.156,Z 1305.741,A 0.000,B 0.000,C 90.000,E1 169.342} C_DIS
LIN {X -0.141,Y -498.934,Z 1305.734,A 0.000,B 0.000,C 90.000,E1 168.173} C_DIS
LIN {X -0.295,Y -497.713,Z 1305.731,A 0.000,B 0.000,C 90.000,E1 167.589} C_DIS
LIN {X 0.050,Y -495.592,Z 1305.726,A 0.000,B 0.000,C 90.000,E1 166.645} C_DIS
LIN {X -0.012,Y -494.053,Z 1305.723,A 0.000,B 0.000,C 90.000,E1 166.047} C_DIS
LIN {X 0.190,Y -490.572,Z 1305.716,A 0.000,B 0.000,C 90.000,E1 164.810} C_DIS
LIN {X -0.007,Y -486.861,Z 1305.709,A 0.000,B 0.000,C 90.000,E1 163.614} C_DIS
LIN {X 0.104,Y -485.098,Z 1305.706,A 0.000,B 0.000,C 90.000,E1 163.142} C_DIS
LIN {X 0.201,Y -482.105,Z 1305.702,A 0.000,B 0.000,C 90.000,E1 162.362} C_DIS
LIN {X 0.031,Y -477.559,Z 1305.697,A 0.000,B 0.000,C 90.000,E1 161.456} C_DIS
LIN {X -0.162,Y -474.512,Z 1305.694,A 0.000,B 0.000,C 90.000,E1 160.859} C_DIS
LIN {X 0.186,Y -470.792,Z 1305.688,A 0.000,B 0.000,C 90.000,E1 159.880} C_DIS
LIN {X 0.106,Y -468.835,Z 1305.685,A 0.000,B 0.000,C 90.000,E1 159.263} C_DIS
LIN {X 0.012,Y -467.648,Z 1305.681,A 0.000,B 0.000,C 90.000,E1 158.646} C_DIS
LIN {X 0.100,Y -467.936,Z 1305.677,A 0.000,B 0.000,C 90.000,E1 157.847} C_DIS
LIN {X -0.143,Y -468.569,Z 1305.676,A 0.000,B 0.000,C 90.000,E1 157.720} C_DIS
LIN {X 0.078,Y -469.608,Z 1305.674,A 0.000,B 0.000,C 90.000,E1 157.358} C_DIS
LIN {X 0.038,Y -469.617,Z 1305.674,A 0.000,B 0.000,C 90.000,E1 157.358} C_DIS
LIN {X 0.189,Y -471.824,Z 1305.673,A 0.000,B 0.000,C 90.000,E1 157.050} C_DIS
LIN {X -0.134,Y -475.175,Z 1305.671,A 0.000,B 0.000,C 90.000,E1 156.794} C_DIS
LIN {X 0.185,Y -477.968,Z 1305.670,A 0.000,B 0.000,C 90.000,E1 156.485} C_DIS
LIN {X -0.091,Y -484.601,Z 1305.667,A 0.000,B 0.000,C 90.000,E1 155.973} C_DIS
LIN {X -0.287,Y -491.990,Z 1305.663,A 0.000,B 0.000,C 90.000,E1 155.357} C_DIS
LIN {X 0.050,Y -499.191,Z 1305.659,A 0.000,B 0.000,C 90.000,E1 154.665} C_DIS
LIN {X -0.194,Y -504.774,Z 1305.656,A 0.000,B 0.000,C 90.000,E1 154.152} C_DIS
LIN {X -0.098,Y -511.264,Z 1305.652,A 0.000,B 0.000,C 90.000,E1 153.435} C_DIS
LIN {X -0.121,Y -515.086,Z 1305.650,A 0.000,B 0.000,C 90.000,E1 152.999} C_DIS
LIN {X -0.088,Y -519.750,Z 1305.647,A 0.000,B 0.000,C 90.000,E1 152.410} C_DIS
LIN {X -0.126,Y -522.976,Z 1305.644,A 0.000,B 0.000,C 90.000,E1 151.975} C_DIS
LIN {X -0.215,Y -527.555,Z 1305.640,A 0.000,B 0.000,C 90.000,E1 151.257} C_DIS
LIN {X -0.112,Y -530.588,Z 1305.637,A 0.000,B 0.000,C 90.000,E1 150.667} C_DIS
LIN {X 0.132,Y -533.690,Z 1305.633,A 0.000,B 0.000,C 90.000,E1 149.921} C_DIS
LIN {X 0.282,Y -535.655,Z 1305.630,A 0.000,B 0.000,C 90.000,E1 149.331} C_DIS
LIN {X -0.017,Y -537.291,Z 1305.627,A 0.000,B 0.000,C 90.000,E1 148.791} C_DIS
LIN {X 0.157,Y -539.373,Z 1305.622,A 0.000,B 0.000,C 90.000,E1 147.916} C_DIS
LIN {X 0.073,Y -541.596,Z 1305.616,A 0.000,B 0.000,C 90.000,E1 146.786} C_DIS
LIN {X 0.136,Y -542.927,Z 1305.611,A 0.000,B 0.000,C 90.000,E1 145.928} C_DIS
LIN {X -0.144,Y -543.830,Z 1305.609,A 0.000,B 0.000,C 90.000,E1 145.674} C_DIS
LIN {X 0.024,Y -544.812,Z 1305.609,A 0.000,B 0.000,C 90.000,E1 145.515} C_DIS
LIN {X -0.200,Y -545.853,Z 1305.608,A 0.000,B 0.000,C 90.000,E1 145.468} C_DIS
LIN {X 0.108,Y -550.365,Z 1305.607,A 0.000,B 0.000,C 90.000,E1 145.182} C_DIS
LIN {X 0.237,Y -559.368,Z 1305.604,A 0.000,B 0.000,C 90.000,E1 144.769} C_DIS
LIN {X 0.018,Y -564.313,Z 1305.603,A 0.000,B 0.000,C 90.000,E1 144.562} C_DIS
LIN {X 0.043,Y -567.305,Z 1305.602,A 0.000,B 0.000,C 90.000,E1 144.402} C_DIS
LIN {X 0.206,Y -576.360,Z 1305.599,A 0.000,B 0.000,C 90.000,E1 143.829} C_DIS
LIN {X -0.102,Y -582.202,Z 1305.597,A 0.000,B 0.000,C 90.000,E1 143.463} C_DIS
LIN {X 0.088,Y -587.768,Z 1305.595,A 0.000,B 0.000,C 90.000,E1 143.004} C_DIS
LIN {X -0.193,Y -591.843,Z 1305.593,A 0.000,B 0.000,C 90.000,E1 142.683} C_DIS
LIN {X -0.138,Y -597.048,Z 1305.590,A 0.000,B 0.000,C 90.000,E1 142.190} C_DIS
LIN {X -0.268,Y -600.736,Z 1305.588,A 0.000,B 0.000,C 90.000,E1 141.823} C_DIS
LIN {X 0.282,Y -605.334,Z 1305.585,A 0.000,B 0.000,C 90.000,E1 141.251} C_DIS
LIN {X 0.339,Y -609.580,Z 1305.582,A 0.000,B 0.000,C 90.000,E1 140.723} C_DIS
LIN {X 0.046,Y -613.512,Z 1305.579,A 0.000,B 0.000,C 90.000,E1 140.231} C_DIS
LIN {X 0.158,Y -617.165,Z 1305.576,A 0.000,B 0.000,C 90.000,E1 139.703} C_DIS
LIN {X 0.023,Y -621.303,Z 1305.573,A 0.000,B 0.000,C 90.000,E1 139.094} C_DIS
LIN {X 0.046,Y -625.851,Z 1305.568,A 0.000,B 0.000,C 90.000,E1 138.324} C_DIS
LIN {X 0.118,Y -630.192,Z 1305.564,A 0.000,B 0.000,C 90.000,E1 137.553} C_DIS
LIN {X 0.165,Y -634.821,Z 1305.559,A 0.000,B 0.000,C 90.000,E1 136.662} C_DIS
LIN {X 0.151,Y -641.165,Z 1305.552,A 0.000,B 0.000,C 90.000,E1 135.405} C_DIS
LIN {X 0.334,Y -645.475,Z 1305.547,A 0.000,B 0.000,C 90.000,E1 134.514} C_DIS
LIN {X 0.006,Y -652.080,Z 1305.540,A 0.000,B 0.000,C 90.000,E1 133.176} C_DIS
LIN {X -0.134,Y -655.605,Z 1305.536,A 0.000,B 0.000,C 90.000,E1 132.447} C_DIS
LIN {X -0.262,Y -661.278,Z 1305.529,A 0.000,B 0.000,C 90.000,E1 131.229} C_DIS
LIN {X 0.168,Y -664.560,Z 1305.525,A 0.000,B 0.000,C 90.000,E1 130.458} C_DIS
LIN {X -0.245,Y -669.588,Z 1305.518,A 0.000,B 0.000,C 90.000,E1 129.277} C_DIS
LIN {X 0.365,Y -674.114,Z 1305.511,A 0.000,B 0.000,C 90.000,E1 128.016} C_DIS
LIN {X 0.081,Y -676.685,Z 1305.507,A 0.000,B 0.000,C 90.000,E1 127.317} C_DIS
LIN {X -0.163,Y -679.785,Z 1305.502,A 0.000,B 0.000,C 90.000,E1 126.377} C_DIS
LIN {X 0.179,Y -682.607,Z 1305.497,A 0.000,B 0.000,C 90.000,E1 125.391} C_DIS
LIN {X -0.005,Y -685.137,Z 1305.491,A 0.000,B 0.000,C 90.000,E1 124.452} C_DIS
LIN {X 0.386,Y -686.889,Z 1305.487,A 0.000,B 0.000,C 90.000,E1 123.706} C_DIS
LIN {X -0.151,Y -688.456,Z 1305.484,A 0.000,B 0.000,C 90.000,E1 123.038} C_DIS
LIN {X -0.080,Y -690.215,Z 1305.478,A 0.000,B 0.000,C 90.000,E1 122.084} C_DIS
LIN {X 0.010,Y -691.820,Z 1305.473,A 0.000,B 0.000,C 90.000,E1 121.131} C_DIS
LIN {X -0.356,Y -693.921,Z 1305.465,A 0.000,B 0.000,C 90.000,E1 119.745} C_DIS
LIN {X 0.365,Y -695.001,Z 1305.460,A 0.000,B 0.000,C 90.000,E1 118.743} C_DIS
LIN {X -0.179,Y -695.797,Z 1305.455,A 0.000,B 0.000,C 90.000,E1 117.847} C_DIS
LIN {X 0.230,Y -696.181,Z 1305.449,A 0.000,B 0.000,C 90.000,E1 116.873} C_DIS
LIN {X 0.071,Y -696.222,Z 1305.446,A 0.000,B 0.000,C 90.000,E1 116.181} C_DIS
LIN {X 0.219,Y -695.976,Z 1305.442,A 0.000,B 0.000,C 90.000,E1 115.463} C_DIS
LIN {X -0.195,Y -695.558,Z 1305.439,A 0.000,B 0.000,C 90.000,E1 115.027} C_DIS
LIN {X 0.314,Y -694.833,Z 1305.436,A 0.000,B 0.000,C 90.000,E1 114.515} C_DIS
LIN {X -0.354,Y -694.382,Z 1305.435,A 0.000,B 0.000,C 90.000,E1 114.335} C_DIS
LIN {X 0.143,Y -692.848,Z 1305.432,A 0.000,B 0.000,C 90.000,E1 113.823} C_DIS
LIN {X 0.110,Y -691.727,Z 1305.431,A 0.000,B 0.000,C 90.000,E1 113.590} C_DIS
LIN {X 0.043,Y -688.886,Z 1305.429,A 0.000,B 0.000,C 90.000,E1 113.131} C_DIS
LIN {X -0.112,Y -687.782,Z 1305.428,A 0.000,B 0.000,C 90.000,E1 113.025} C_DIS
LIN {X 0.272,Y -684.748,Z 1305.427,A 0.000,B 0.000,C 90.000,E1 112.770} C_DIS
LIN {X 0.253,Y -681.204,Z 1305.425,A 0.000,B 0.000,C 90.000,E1 112.514} C_DIS
LIN {X -0.334,Y -678.899,Z 1305.425,A 0.000,B 0.000,C 90.000,E1 112.461} C_DIS
LIN {X -0.117,Y -674.191,Z 1305.424,A 0.000,B 0.000,C 90.000,E1 112.280} C_DIS
LIN {X 0.053,Y -672.230,Z 1305.423,A 0.000,B 0.000,C 90.000,E1 112.206} C_DIS
LIN {X -0.056,Y -663.749,Z 1305.423,A 0.000,B 0.000,C 90.000,E1 112.078} C_DIS
LIN {X 0.010,Y -657.247,Z 1305.422,A 0.000,B 0.000,C 90.000,E1 112.025} C_DIS
LIN {X -0.329,Y -649.934,Z 1305.422,A 0.000,B 0.000,C 90.000,E1 112.025} C_DIS
LIN {X -0.134,Y -644.441,Z 1305.422,A 0.000,B 0.000,C 90.000,E1 111.950} C_DIS
LIN {X 0.083,Y -641.601,Z 1305.421,A 0.000,B 0.000,C 90.000,E1 111.844} C_DIS
LIN {X 0.042,Y -641.570,Z 1305.421,A 0.000,B 0.000,C 90.000,E1 111.844} C_DIS
LIN {X -0.119,Y -643.145,Z 1305.420,A 0.000,B 0.000,C 90.000,E1 111.535} C_DIS
LIN {X -0.152,Y -650.930,Z 1305.414,A 0.000,B 0.000,C 90.000,E1 110.536} C_DIS
LIN {X 0.216,Y -655.190,Z 1305.411,A 0.000,B 0.000,C 90.000,E1 109.885} C_DIS
LIN {X 0.282,Y -659.486,Z 1305.406,A 0.000,B 0.000,C 90.000,E1 109.141} C_DIS
LIN {X 0.061,Y -662.069,Z 1305.404,A 0.000,B 0.000,C 90.000,E1 108.671} C_DIS
LIN {X -0.028,Y -665.347,Z 1305.400,A 0.000,B 0.000,C 90.000,E1 107.946} C_DIS
LIN {X -0.089,Y -668.269,Z 1305.396,A 0.000,B 0.000,C 90.000,E1 107.221} C_DIS
LIN {X -0.053,Y -669.950,Z 1305.393,A 0.000,B 0.000,C 90.000,E1 106.732} C_DIS
LIN {X -0.266,Y -672.127,Z 1305.389,A 0.000,B 0.000,C 90.000,E1 106.024} C_DIS
LIN {X 0.375,Y -673.924,Z 1305.385,A 0.000,B 0.000,C 90.000,E1 105.245} C_DIS
LIN {X 0.206,Y -675.430,Z 1305.381,A 0.000,B 0.000,C 90.000,E1 104.537} C_DIS
LIN {X 0.054,Y -676.707,Z 1305.377,A 0.000,B 0.000,C 90.000,E1 103.828} C_DIS
LIN {X -0.089,Y -677.574,Z 1305.373,A 0.000,B 0.000,C 90.000,E1 103.119} C_DIS
LIN {X -0.181,Y -677.943,Z 1305.370,A 0.000,B 0.000,C 90.000,E1 102.647} C_DIS
LIN {X 0.205,Y -678.163,Z 1305.366,A 0.000,B 0.000,C 90.000,E1 101.895} C_DIS
LIN {X 0.117,Y -678.115,Z 1305.364,A 0.000,B 0.000,C 90.000,E1 101.422} C_DIS
LIN {X 0.025,Y -677.883,Z 1305.361,A 0.000,B 0.000,C 90.000,E1 100.950} C_DIS
LIN {X -0.245,Y -677.145,Z 1305.357,A 0.000,B 0.000,C 90.000,E1 100.254} C_DIS
LIN {X 0.316,Y -676.431,Z 1305.354,A 0.000,B 0.000,C 90.000,E1 99.726} C_DIS
LIN {X 0.091,Y -675.369,Z 1305.352,A 0.000,B 0.000,C 90.000,E1 99.265} C_DIS
LIN {X -0.137,Y -673.995,Z 1305.349,A 0.000,B 0.000,C 90.000,E1 98.803} C_DIS
LIN {X -0.271,Y -672.199,Z 1305.346,A 0.000,B 0.000,C 90.000,E1 98.333} C_DIS
LIN {X -0.023,Y -669.055,Z 1305.342,A 0.000,B 0.000,C 90.000,E1 97.587} C_DIS
LIN {X 0.097,Y -663.945,Z 1305.337,A 0.000,B 0.000,C 90.000,E1 96.606} C_DIS
LIN {X -0.222,Y -660.412,Z 1305.333,A 0.000,B 0.000,C 90.000,E1 96.024} C_DIS
LIN {X 0.013,Y -656.322,Z 1305.330,A 0.000,B 0.000,C 90.000,E1 95.391} C_DIS
LIN {X 0.261,Y -652.821,Z 1305.327,A 0.000,B 0.000,C 90.000,E1 94.878} C_DIS
LIN {X -0.214,Y -647.903,Z 1305.324,A 0.000,B 0.000,C 90.000,E1 94.302} C_DIS
LIN {X 0.031,Y -643.660,Z 1305.321,A 0.000,B 0.000,C 90.000,E1 93.784} C_DIS
LIN {X -0.126,Y -635.608,Z 1305.316,A 0.000,B 0.000,C 90.000,E1 92.922} C_DIS
LIN {X -0.206,Y -628.372,Z 1305.312,A 0.000,B 0.000,C 90.000,E1 92.178} C_DIS
LIN {X 0.055,Y -623.373,Z 1305.309,A 0.000,B 0.000,C 90.000,E1 91.661} C_DIS
LIN {X -0.122,Y -616.508,Z 1305.306,A 0.000,B 0.000,C 90.000,E1 91.088} C_DIS
LIN {X 0.226,Y -609.005,Z 1305.303,A 0.000,B 0.000,C 90.000,E1 90.516} C_DIS
LIN {X 0.239,Y -602.573,Z 1305.301,A 0.000,B 0.000,C 90.000,E1 90.115} C_DIS
LIN {X 0.031,Y -595.822,Z 1305.299,A 0.000,B 0.000,C 90.000,E1 89.771} C_DIS
LIN {X 0.236,Y -588.592,Z 1305.297,A 0.000,B 0.000,C 90.000,E1 89.427} C_DIS
LIN {X 0.138,Y -576.010,Z 1305.294,A 0.000,B 0.000,C 90.000,E1 88.969} C_DIS
LIN {X 0.093,Y -572.124,Z 1305.293,A 0.000,B 0.000,C 90.000,E1 88.797} C_DIS
LIN {X 0.045,Y -572.042,Z 1305.293,A 0.000,B 0.000,C 90.000,E1 88.797} C_DIS
LIN {X -0.251,Y -570.365,Z 1305.292,A 0.000,B 0.000,C 90.000,E1 88.568} C_DIS
LIN {X 0.276,Y -570.338,Z 1305.292,A 0.000,B 0.000,C 90.000,E1 88.511} C_DIS
LIN {X -0.019,Y -570.107,Z 1305.290,A 0.000,B 0.000,C 90.000,E1 88.224} C_DIS
LIN {X -0.113,Y -571.299,Z 1305.281,A 0.000,B 0.000,C 90.000,E1 86.674} C_DIS
LIN {X 0.049,Y -573.847,Z 1305.268,A 0.000,B 0.000,C 90.000,E1 84.204} C_DIS
LIN {X -0.259,Y -575.364,Z 1305.260,A 0.000,B 0.000,C 90.000,E1 82.875} C_DIS
LIN {X 0.243,Y -577.321,Z 1305.251,A 0.000,B 0.000,C 90.000,E1 81.197} C_DIS
LIN {X 0.202,Y -579.251,Z 1305.242,A 0.000,B 0.000,C 90.000,E1 79.577} C_DIS
LIN {X 0.181,Y -580.670,Z 1305.235,A 0.000,B 0.000,C 90.000,E1 78.229} C_DIS
LIN {X -0.042,Y -581.703,Z 1305.229,A 0.000,B 0.000,C 90.000,E1 77.173} C_DIS
LIN {X -0.022,Y -582.808,Z 1305.221,A 0.000,B 0.000,C 90.000,E1 75.825} C_DIS
LIN {X -0.080,Y -583.610,Z 1305.215,A 0.000,B 0.000,C 90.000,E1 74.755} C_DIS
LIN {X -0.059,Y -584.662,Z 1305.206,A 0.000,B 0.000,C 90.000,E1 73.142} C_DIS
LIN {X 0.163,Y -585.706,Z 1305.197,A 0.000,B 0.000,C 90.000,E1 71.511} C_DIS
LIN {X -0.144,Y -586.723,Z 1305.188,A 0.000,B 0.000,C 90.000,E1 69.934} C_DIS
LIN {X 0.317,Y -587.776,Z 1305.180,A 0.000,B 0.000,C 90.000,E1 68.284} C_DIS
LIN {X -0.304,Y -588.830,Z 1305.171,A 0.000,B 0.000,C 90.000,E1 66.741} C_DIS
LIN {X 0.105,Y -589.904,Z 1305.162,A 0.000,B 0.000,C 90.000,E1 65.101} C_DIS
LIN {X 0.006,Y -591.029,Z 1305.153,A 0.000,B 0.000,C 90.000,E1 63.512} C_DIS
LIN {X 0.098,Y -592.552,Z 1305.143,A 0.000,B 0.000,C 90.000,E1 61.641} C_DIS
LIN {X -0.109,Y -593.870,Z 1305.135,A 0.000,B 0.000,C 90.000,E1 60.333} C_DIS
LIN {X 0.118,Y -595.719,Z 1305.125,A 0.000,B 0.000,C 90.000,E1 58.456} C_DIS
LIN {X -0.114,Y -597.691,Z 1305.115,A 0.000,B 0.000,C 90.000,E1 56.628} C_DIS
LIN {X 0.126,Y -599.333,Z 1305.106,A 0.000,B 0.000,C 90.000,E1 55.022} C_DIS
LIN {X -0.084,Y -600.818,Z 1305.097,A 0.000,B 0.000,C 90.000,E1 53.463} C_DIS
LIN {X -0.273,Y -602.187,Z 1305.088,A 0.000,B 0.000,C 90.000,E1 51.904} C_DIS
LIN {X 0.301,Y -603.323,Z 1305.079,A 0.000,B 0.000,C 90.000,E1 50.275} C_DIS
LIN {X -0.209,Y -604.233,Z 1305.072,A 0.000,B 0.000,C 90.000,E1 49.013} C_DIS
LIN {X -0.116,Y -604.550,Z 1305.066,A 0.000,B 0.000,C 90.000,E1 47.957} C_DIS
LIN {X 0.187,Y -604.800,Z 1305.059,A 0.000,B 0.000,C 90.000,E1 46.620} C_DIS
LIN {X -0.131,Y -604.898,Z 1305.050,A 0.000,B 0.000,C 90.000,E1 45.081} C_DIS
LIN {X -0.056,Y -604.730,Z 1305.045,A 0.000,B 0.000,C 90.000,E1 44.028} C_DIS
LIN {X 0.255,Y -604.414,Z 1305.037,A 0.000,B 0.000,C 90.000,E1 42.690} C_DIS
